	16#4B7A: sMsg := '4B7A function not implemented';
	16#4B7B: sMsg := '4B7B parameter Tangential Following: The radius of the actual circle segment is too small';
	16#4B7C: sMsg := '4B7C parameter FB_NciFeedTablePreparation: pEntry is NULL';
	16#4B7D: sMsg := '4B7D parameter FB_NciFeedTablePreparation: The specified nEntryType does not match the the structure type';
	16#4B7E: sMsg := '4B7E parameter ST_NciMFuncFast and ST_NciMFuncHsk: The requested m-function is not in between 0..159';
	16#4B7F: sMsg := '4B7F parameter ST_NciDynOvr: The requested value for the dynamic override is not in between 0.01 and 1.0';
	16#4B80: sMsg := '4B80 parameter ST_NciVertexSmoothing: invalid parameter. This error occurs with a negative vertex radius or an unknown vertex smoothing type.';
	16#4B81: sMsg := '4B81 parameter FB_NciFeedTablePrepartion: The requested velocity is not in a valid range';
	16#4B82: sMsg := '4B82 parameter ST_Nci*: invalid parameter';

ELSE
	sMsg := UDINT_TO_STRING(iErrID);
	sMsg := concat(sMsg, ' Unknown Error code');
END_CASE
F_AxErrMsg := sMsg;

END_FUNCTION

// ---- POUs/FB/AxisControl/Internal/HomingAdv/FB_HomingLimitSwitch.TcPOU
//==================================================================================================
//							Beckhoff Automation Poland
//									3.01.2022
//	Function block running PLC CAM procedure using hardware limit switch
//	Library: Tc3_MC2_AdvancedHoming, Tc2_MC2, 
//
//  v1.0	|| TC v 3.1.4024.22		|| First edition 
//==================================================================================================
FUNCTION_BLOCK FB_HomingLimitSwitch
VAR_IN_OUT
	Axis 										: Tc2_MC2.AXIS_REF;
END_VAR
VAR_INPUT
	bExecute									: BOOL;
	eDirection									: Tc3_MC2_AdvancedHoming.MC_Home_Direction;
	eLimitSwitchMode							: Tc3_MC2_AdvancedHoming.MC_Switch_Mode;
	eLimitSwitchSignal							: Tc3_MC2_AdvancedHoming.MC_Ref_Signal_Ref;
	lrVelocity									: LREAL;
	lrSetPosition								: LREAL;
	tTimeLimit									: TIME;
	lrDistanceLimit								: LREAL;
	lrTorqueLimit								: LREAL;
	lrDistance									: LREAL;
END_VAR                             		
VAR_OUTPUT                              		
	bDone										: BOOL;
	bBusy										: BOOL;
	bCommandAborted								: BOOL;
	bError										: BOOL;
	nErrorID									: UDINT;
END_VAR
VAR
//=========================== Common ============================
	nStep										: UDINT;
	stParameter									: Tc3_MC2_AdvancedHoming.MC_HomingParameter;
	stOptions									: Tc3_MC2_AdvancedHoming.ST_Home_Options4;
	mcStepLimitSwitch							: Tc3_MC2_AdvancedHoming.MC_StepLimitSwitch;
//=========================== Finish ============================
	mcFinishHoming								: Tc3_MC2_AdvancedHoming.MC_FinishHoming;
//============================ Abort ============================
	mcAbortHoming								: Tc3_MC2_AdvancedHoming.MC_AbortHoming;
//========================== Internal ===========================
    {attribute 'hide'}
	nErrorID_Int								: UDINT;
//===============================================================
END_VAR

//====== Call FBs outside CASE - easier debugging ===============
mcStepLimitSwitch(	Axis						:= Axis, 
					Parameter					:= stParameter,
					LimitSwitchMode				:= eLimitSwitchMode, 
					LimitSwitchSignal			:= eLimitSwitchSignal);
                                        		
mcFinishHoming(	Axis							:= Axis, 
				Parameter						:= stParameter);
				                        	
mcAbortHoming(	Axis							:= Axis, 
				Parameter						:= stParameter);
				
//============== CASE instruction - step machine ================
CASE nStep OF
	
	0: // Wait for command
	
		IF bExecute THEN
			bBusy								:= TRUE;
				
			mcStepLimitSwitch(	Axis			:= Axis, 
								Parameter		:= stParameter,
								Execute			:= TRUE,
								Direction		:= eDirection,  
								Velocity		:= lrVelocity,
								SetPosition		:= lrSetPosition, 
								TimeLimit		:= tTimeLimit, 
								DistanceLimit	:= lrDistanceLimit,
								TorqueLimit		:= lrTorqueLimit,  
								Options			:= stOptions);
								
			// Latch finish parameters
			mcFinishHoming.Distance				:= lrDistance;
			mcFinishHoming.Velocity				:= lrVelocity;
						
			nStep								:= 1000;

		END_IF
	
	1000: // Wait till end
	
		IF mcStepLimitSwitch.Done THEN
			mcStepLimitSwitch.Execute			:= FALSE;
			nStep 								:= 3000;
		END_IF
		
		IF mcStepLimitSwitch.CommandAborted THEN
			mcStepLimitSwitch.Execute			:= FALSE;
			bBusy 								:= FALSE;
			bCommandAborted						:= TRUE;
			nStep 								:= 6000;
		END_IF
		
		IF mcStepLimitSwitch.Error THEN
			mcStepLimitSwitch.Execute			:= FALSE;
			nErrorID_Int						:= mcStepLimitSwitch.ErrorID;
			nStep 								:= 4000;
		END_IF
		
	3000: // MC_FinishHoming
	
		mcFinishHoming.Execute					:= TRUE;				
		nStep									:= nStep + 10;
		
	3010: // Wait till end
	
		IF mcFinishHoming.Done THEN
			mcFinishHoming.Execute				:= FALSE;
			bBusy 								:= FALSE;
			bDone 								:= TRUE;
			nStep 								:= 5000;
		END_IF
		
		IF mcFinishHoming.CommandAborted THEN
			mcFinishHoming.Execute				:= FALSE;
			bBusy 								:= FALSE;
			bCommandAborted						:= TRUE;
			nStep 								:= 6000;
		END_IF
		
		IF mcFinishHoming.Error THEN
			mcFinishHoming.Execute				:= FALSE;
			bBusy 								:= FALSE;
			bError								:= TRUE;
			nErrorID							:= mcFinishHoming.ErrorID;
			nStep 								:= 10000;
		END_IF	
		
	4000: // MC_AbortHoming
	
		mcAbortHoming.Execute					:= TRUE;				
		nStep									:= nStep + 10;
		
	4010: // Wait till end
	
		// No matter what is the end, we go to error State
		IF NOT mcAbortHoming.Busy THEN
			mcAbortHoming.Execute				:= FALSE;
			bBusy 								:= FALSE;
			bError								:= TRUE;
			nErrorID							:= nErrorID_Int;			
			nStep								:= 10000;
		END_IF
		
	5000: // Done
	
		bDone									:= bExecute;
		IF NOT bExecute THEN
			nStep 								:= 0;
		END_IF	
	
	6000: // Command Aborted
	
		bCommandAborted							:= bExecute;
		IF NOT bExecute THEN
			nStep 								:= 0;
		END_IF
		
	10000..20000: // Error
	
		bError									:= bExecute;
		IF NOT bExecute THEN
			nErrorID							:= 0;
			nErrorID_Int						:= 0;
			nStep 								:= 0;
		END_IF
		
END_CASE
//===============================================================

END_FUNCTION_BLOCK

// ---- POUs/FB/AxisControl/Internal/HomingAdv/FB_HomingMemoryAX8000.TcPOU
//==================================================================================================
//							Beckhoff Automation Poland
//									3.01.2022
//	Function block running PLC CAM procedure and writes offset to encoder memory via AX8000
//	During procedure there is need to enable/disable power - external handling needed
//	Velocity to and off cam and moving direction taken from NC Axis settings
//	Library: Tc2_MC2, Tc2_MC2_Drive, Tc2_System
//
//  v1.0	|| TC v 3.1.4024.22		|| First edition 
//==================================================================================================
FUNCTION_BLOCK FB_HomingMemoryAX8000
VAR_IN_OUT                              		
	Axis										: AXIS_REF;
END_VAR  
VAR_INPUT
	bExecute									: BOOL;								// Rising edge executes cmd
	lrPosition									: LREAL;
	eHomingMode									: Tc2_MC2.MC_HomingMode;
	eFeedback									: Tc2_MC2_Drive.E_PositionOffsetFeedback;
	eMemory										: Tc2_MC2_Drive.E_PositionOffsetMemory;
	bCalibrationCam								: BOOL;
	bPowerStatus								: BOOL;								// 
END_VAR                               		
VAR_OUTPUT                              		
	bDone										: BOOL;
	bBusy										: BOOL;
	bCommandAborted								: BOOL;
	bError										: BOOL;
	nErrorID									: UDINT;
	bEnablePower								: BOOL;
END_VAR                                 		
VAR
	// =================================== Local ======================================
	nStep										: DINT;				// Case step
	lrLatchPos									: LREAL;			// Last latched position - cam falling edge
	// ================================ Internal hidden ===============================
    {attribute 'hide'}
	lrPositionMem								: LREAL;
    {attribute 'hide'}
	eHomingModeMem								: Tc2_MC2.MC_HomingMode;
    {attribute 'hide'}
	eFeedbackMem								: Tc2_MC2_Drive.E_PositionOffsetFeedback;
    {attribute 'hide'}
	eMemoryMem									: Tc2_MC2_Drive.E_PositionOffsetMemory;
    {attribute 'hide'}
	lrOffs										: LREAL;
    {attribute 'hide'}
	lrVelocityTw								: LREAL;			// 40xx/6
    {attribute 'hide'}
	lrVelocityOff								: LREAL;			// 40xx/7
    {attribute 'hide'}
	wInvertDirection							: WORD;				// 50xx/101
	// ===================================== FBs ======================================
    {attribute 'hide'}
	fbADSREAD									: ADSREAD;
    {attribute 'hide'}
	mcHome										: MC_Home;
    {attribute 'hide'}
	mcHalt										: MC_Halt;	
    {attribute 'hide'}
	mcReset										: MC_Reset;	
    {attribute 'hide'}
	mcMoveVelocity								: MC_MoveVelocity;
    {attribute 'hide'}
	fbDeletePositionOffset						: FB_CoEAX8000DeletePositionOffset;
    {attribute 'hide'}
	fbSetPositionOffset							: FB_CoEAX8000SetPositionOffset;
	// ================================================================================
END_VAR

fbDeletePositionOffset(Axis:= Axis);
fbSetPositionOffset(Axis:= Axis);
	
mcMoveVelocity(Axis:= Axis);	
mcHalt(Axis:= Axis);
mcHome(Axis := Axis);
mcReset(Axis:= Axis);

CASE nStep OF
	
	0: // Wait for command
	
		IF bExecute THEN
			lrPositionMem						:= lrPosition;
			eHomingModeMem						:= eHomingMode;
			eFeedbackMem						:= eFeedback;
			eMemoryMem							:= eMemory;
			bBusy								:= TRUE;
			nStep 								:= nStep + 10;
		END_IF

	10: // MC_HomingMode.MC_ResetCalibration - All types need it
	
		mcHome.Execute							:= TRUE;
		mcHome.HomingMode						:= MC_HomingMode.MC_ResetCalibration;
		nStep 									:= nStep + 10;

	20: // Wait till end
	
		IF mcHome.Done THEN
			mcHome.Execute						:= FALSE;
			// Next step depends on homing type
			IF eHomingModeMem = MC_HomingMode.MC_ResetCalibration THEN
				bBusy 							:= FALSE;
				bDone							:= TRUE;
				nStep 							:= 5000;
			END_IF
			
			IF eHomingModeMem = MC_HomingMode.MC_DefaultHoming THEN
				nStep							:= 1000;
			END_IF
	
			IF eHomingModeMem = MC_HomingMode.MC_Direct THEN
				nStep							:= 2000;
			END_IF
	
			IF eHomingModeMem = MC_HomingMode.MC_ForceCalibration THEN
				nStep							:= 3000;
			END_IF

		END_IF
		
		IF mcHome.CommandAborted THEN
			mcHome.Execute						:= FALSE;
			bBusy 								:= FALSE;
			bCommandAborted						:= TRUE;
			nStep 								:= 6000;
		END_IF
		
		IF mcHome.Error THEN
			mcHome.Execute						:= FALSE;
			nErrorID							:= mcHome.ErrorID;
			bBusy 								:= FALSE;
			bError								:= TRUE;
			nStep 								:= nStep + 10000;
		END_IF
		
	1000, 2000: // First remove existing position offset

		IF NOT bPowerStatus THEN
			fbDeletePositionOffset.Execute		:= TRUE;
			fbDeletePositionOffset.Feedback		:= eFeedbackMem;
			fbDeletePositionOffset.Memory		:= eMemoryMem;
			nStep 								:= nStep + 10;
		END_IF
		
	1010, 2010: // Wait till command end
	
		IF NOT fbDeletePositionOffset.Busy THEN
			fbDeletePositionOffset.Execute		:= FALSE;
			IF fbDeletePositionOffset.Error THEN
				nErrorID						:= fbDeletePositionOffset.ErrorID;
				bBusy 							:= FALSE;
				bError							:= TRUE;
				nStep 							:= nStep + 10000;
			ELSE
				nStep 							:= nStep + 10;
			END_IF
		END_IF

	1020: // Write 0 offs - to make moves possible
	
		fbSetPositionOffset.Execute				:= TRUE;
		fbSetPositionOffset.Relative			:= TRUE;
		fbSetPositionOffset.Position			:= 0;
		fbSetPositionOffset.Feedback			:= eFeedbackMem;
		fbSetPositionOffset.Memory				:= eMemoryMem;
		nStep 									:= nStep + 10;		
	
	1030:  // Wait till command end
	
		IF NOT fbSetPositionOffset.Busy THEN
			fbSetPositionOffset.Execute		:= FALSE;
			IF fbSetPositionOffset.Error THEN
				nErrorID						:= fbSetPositionOffset.ErrorID;
				bBusy 							:= FALSE;
				bError							:= TRUE;
				nStep 							:= nStep + 10000;
			ELSE
				nStep 							:=  nStep + 10;	
			END_IF
		END_IF

	1040: // Read lrVelocityTw
	
		fbADSREAD(	READ		:= TRUE,
					NETID		:= '', 
					PORT		:= 500,
					IDXGRP		:= 16#4000 + Axis.NcToPlc.AxisId,
					IDXOFFS		:= 16#0006,
					LEN			:= SIZEOF(lrVelocityTw), 
					DESTADDR	:= ADR(lrVelocityTw));
		
		nStep 									:= nStep + 10;

	1060: // Read lrVelocityOff
	
		fbADSREAD(	READ		:= TRUE,
					NETID		:= '', 
					PORT		:= 500,
					IDXGRP		:= 16#4000 + Axis.NcToPlc.AxisId,
					IDXOFFS		:= 16#0007,
					LEN			:= SIZEOF(lrVelocityOff), 
					DESTADDR	:= ADR(lrVelocityOff));
		
		nStep 									:= nStep + 10;
		
	1080: // Read bInvertDirection
	
		fbADSREAD(	READ		:= TRUE,
					NETID		:= '', 
					PORT		:= 500,
					IDXGRP		:= 16#5000 + Axis.NcToPlc.AxisId,
					IDXOFFS		:= 16#0101,
					LEN			:= SIZEOF(wInvertDirection), 
					DESTADDR	:= ADR(wInvertDirection));
		
		nStep 									:= nStep + 10;
	
	1050,1070,1090:  // Wait till command end
	
		fbADSREAD();
		IF NOT fbADSREAD.BUSY THEN
			IF NOT fbADSREAD.ERR THEN
				fbADSREAD(READ:= FALSE);
				nStep 							:= nStep + 10;
			ELSE
				nErrorID						:= fbADSREAD.ERRID;
				bBusy							:= FALSE;
				bError							:= TRUE;
				fbADSREAD(READ:= FALSE);
				nStep 							:= nStep + 10000;	
			END_IF
		END_IF

	1100: // Reset AX8000 offset error
	
		mcReset.Execute							:= TRUE;
		nStep 									:= nStep + 10;

	1110: // Wait till command end	
	
		IF mcReset.Done THEN
			mcReset.Execute						:= FALSE;
			nStep 								:= nStep + 10;
		END_IF
		
		IF mcReset.Error THEN
			mcReset.Execute						:= FALSE;
			nErrorID							:= mcReset.ErrorID;
			bBusy 								:= FALSE;
			bError								:= TRUE;
			nStep 								:= nStep + 10000;
		END_IF	

	1120: // Enable Power request
	
		bEnablePower							:= TRUE;
		nStep 									:= nStep + 10;
		
	1130: // Power status OK?
	
		IF bPowerStatus THEN
			nStep 								:= nStep + 10;	
		END_IF
	
	1140: // Move velocity to calibration cam
	
		IF wInvertDirection.0 THEN
			mcMoveVelocity.Direction			:= MC_Direction.MC_Negative_Direction;
		ELSE
			mcMoveVelocity.Direction			:= MC_Direction.MC_Positive_Direction;
		END_IF
		mcMoveVelocity.Velocity					:= lrVelocityTw;
		mcMoveVelocity.Execute					:= TRUE;
		nStep 									:= nStep + 10;
	
	1150: // Wait till calibration cam rising edge 
	
		IF bCalibrationCam THEN
			mcMoveVelocity.Execute				:= FALSE;
			nStep 								:= nStep + 10;
		END_IF
		
		IF mcMoveVelocity.CommandAborted THEN
			mcMoveVelocity.Execute				:= FALSE;
			bBusy 								:= FALSE;
			bCommandAborted						:= TRUE;
			nStep 								:= 6000;
		END_IF
		
		IF mcMoveVelocity.Error THEN
			mcMoveVelocity.Execute				:= FALSE;
			nErrorID							:= mcMoveVelocity.ErrorID;
			bBusy 								:= FALSE;
			bError								:= TRUE;
			nStep 								:= nStep + 10000;
		END_IF

	1160: // Halt
	
		mcHalt.Execute							:= TRUE;
		nStep 									:= nStep + 10;
		
	1170:  // Wait till command end
	
		IF mcHalt.Done THEN
			mcHalt.Execute						:= FALSE;
			nStep 								:= nStep + 10;
		END_IF
		
		IF mcHalt.CommandAborted THEN
			mcHalt.Execute						:= FALSE;
			bBusy 								:= FALSE;
			bCommandAborted						:= TRUE;
			nStep 								:= 6000;
		END_IF
		
		IF mcHalt.Error THEN
			mcHalt.Execute						:= FALSE;
			nErrorID							:= mcHalt.ErrorID;
			bBusy 								:= FALSE;
			bError								:= TRUE;
			nStep 								:= nStep + 10000;
		END_IF
		
	1180: // Reference cam became free too soon - ErrorID: 16979
	
		IF NOT bCalibrationCam THEN
			nErrorID							:= 16979;
			bBusy 								:= FALSE;
			bError								:= TRUE;
			nStep 								:= nStep + 10000;
		ELSE
			nStep 								:= nStep + 10;
		END_IF
	
	1190: // Move velocity off calibration cam
	
		IF wInvertDirection.0 THEN
			mcMoveVelocity.Direction			:= MC_Direction.MC_Positive_Direction;
		ELSE
			mcMoveVelocity.Direction			:= MC_Direction.MC_Negative_Direction;
		END_IF
		mcMoveVelocity.Velocity					:= lrVelocityOff;
		mcMoveVelocity.Execute					:= TRUE;
		nStep 									:= nStep + 10;
	
	1200: // Wait till calibration cam falling edge 
	
		IF NOT bCalibrationCam THEN
			lrLatchPos 							:= Axis.NcToPlc.ActPos;
			mcMoveVelocity.Execute				:= FALSE;
			nStep 								:= nStep + 10;
		END_IF
		
		IF mcMoveVelocity.CommandAborted THEN
			mcMoveVelocity.Execute				:= FALSE;
			bBusy 								:= FALSE;
			bCommandAborted						:= TRUE;
			nStep 								:= 6000;
		END_IF
		
		IF mcMoveVelocity.Error THEN
			mcMoveVelocity.Execute				:= FALSE;
			nErrorID							:= mcMoveVelocity.ErrorID;
			bBusy 								:= FALSE;
			bError								:= TRUE;
			nStep 								:= nStep + 10000;
		END_IF

	1210: // Halt
	
		mcHalt.Execute							:= TRUE;
		nStep 									:= nStep + 10;
		
	1220:  // Wait till command end
	
		IF mcHalt.Done THEN
			mcHalt.Execute						:= FALSE;
			nStep 								:= nStep + 10;
		END_IF
		
		IF mcHalt.CommandAborted THEN
			mcHalt.Execute						:= FALSE;
			bBusy 								:= FALSE;
			bCommandAborted						:= TRUE;
			nStep 								:= 6000;
		END_IF
		
		IF mcHalt.Error THEN
			mcHalt.Execute						:= FALSE;
			nErrorID							:= mcHalt.ErrorID;
			bBusy 								:= FALSE;
			bError								:= TRUE;
			nStep 								:= nStep + 10000;
		END_IF
		
	1230: // Disable Power request
	
		bEnablePower							:= FALSE;
		nStep 									:= nStep + 10;
		
	1240: // Power status OK?
	
		IF NOT bPowerStatus THEN
			nStep 								:= nStep + 10;	
		END_IF		
	
	1250: // Write pos
	
		lrOffs 									:= lrLatchPos - Axis.NcToPlc.ActPos;
		fbSetPositionOffset.Execute				:= TRUE;
		fbSetPositionOffset.Relative			:= FALSE;
		fbSetPositionOffset.Position			:= lrPositionMem - lrOffs;
		fbSetPositionOffset.Feedback			:= eFeedbackMem;
		fbSetPositionOffset.Memory				:= eMemoryMem;
		nStep 									:= nStep + 10;
		
	1260:  // Wait till command end
	
		IF NOT fbSetPositionOffset.Busy THEN
			fbSetPositionOffset.Execute		:= FALSE;
			IF fbSetPositionOffset.Error THEN
				nErrorID						:= fbSetPositionOffset.ErrorID;
				bBusy 							:= FALSE;
				bError							:= TRUE;
				nStep 							:= nStep + 10000;
			ELSE
				nStep 							:= 3000;		// Set home flag
			END_IF
		END_IF
			
	2020: // Write pos
	
		fbSetPositionOffset.Execute				:= TRUE;
		fbSetPositionOffset.Relative			:= FALSE;
		fbSetPositionOffset.Position			:= lrPositionMem;
		fbSetPositionOffset.Feedback			:= eFeedbackMem;
		fbSetPositionOffset.Memory				:= eMemoryMem;
		nStep 									:= nStep + 10;
		
	2030:  // Wait till command end
	
		IF NOT fbSetPositionOffset.Busy THEN
			fbSetPositionOffset.Execute		:= FALSE;
			IF fbSetPositionOffset.Error THEN
				nErrorID						:= fbSetPositionOffset.ErrorID;
				bBusy 							:= FALSE;
				bError							:= TRUE;
				nStep 							:= nStep + 10000;
			ELSE
				nStep 							:= 3000;		// Set home flag
			END_IF
		END_IF
		
	3000: // MC_HomingMode.MC_ForceCalibration
	
		mcHome.Execute							:= TRUE;
		mcHome.HomingMode						:= MC_HomingMode.MC_ForceCalibration;
		nStep 									:= nStep + 10;

	3010: // Wait till end
	
		IF mcHome.Done THEN
			mcHome.Execute						:= FALSE;
			bBusy 								:= FALSE;
			bDone								:= TRUE;
			nStep 								:= 5000;
		END_IF
		
		IF mcHome.CommandAborted THEN
			bBusy 								:= FALSE;
			bCommandAborted						:= TRUE;
			nStep 								:= 6000;
		END_IF
		
		IF mcHome.Error THEN
			nErrorID							:= mcHome.ErrorID;
			bBusy 								:= FALSE;
			bError								:= TRUE;
			nStep 								:= nStep + 10000;
		END_IF
		
	5000: // Done
	
		bDone									:= bExecute;
		IF NOT bExecute THEN
			nStep 								:= 0;
		END_IF
		
	6000: // Command Aborted
	
		bCommandAborted							:= bExecute;
		IF NOT bExecute THEN
			nStep 								:= 0;
		END_IF
		
	10000..20000: // Error
	
		bError									:= bExecute;
		IF NOT bExecute THEN
			nErrorID							:= 0;
			nStep 								:= 0;
		END_IF
		
END_CASE

END_FUNCTION_BLOCK

// ---- POUs/FB/AxisControl/Internal/HomingAdv/FB_HomingTorqueDetectionSensor.TcPOU
//==================================================================================================
//							Beckhoff Automation Poland
//									3.01.2022
//	Function block running home procedure in torque mode detection
//	Additional sensor can be used
//	Avaliable two modes:
//	1. Lag based - bLagBased = TRUE - define lrLagLimit which decides about end of movement
//	2. Torque based - bLagBased = FALSE - define lrTorqueLimit and lrTorqueTolerance which decides about end of movement
//
//	Library: Tc3_MC2_AdvancedHoming, Tc2_MC2, 
//
//  v1.1	|| TC v 3.1.4024.22		|| Comments added
//  v1.0	|| TC v 3.1.4024.22		|| First edition 
//==================================================================================================
FUNCTION_BLOCK FB_HomingTorqueDetectionSensor
VAR_IN_OUT
	Axis 										: Tc2_MC2.AXIS_REF;
END_VAR  
VAR_INPUT
	bExecute									: BOOL;					// The command is executed with a rising edge.
	bLagBased									: BOOL;					// TRUE: MC_StepBlockLagBased, FALSE: MC_StepBlock
	eDirection									: Tc3_MC2_AdvancedHoming.MC_Home_Direction;	// 
	lrVelocity									: LREAL;				// Maximum travel velocity (>0)
	lrSetPosition								: LREAL;				// Position value to which the axis position is to be set. 
	lrDetectionVelocityLimit					: LREAL;				// Velocity that must be fallen below for the time DetectionVelocityTime in order to detect driving against the fixed stop.
	tDetectionVelocityTime						: TIME;					// Time for detecting the velocity undershoot when driving against the fixed stop.
	tTimeLimit									: TIME;					// Exceeding this time leads to the search procedure being aborted.
	lrDistanceLimit								: LREAL;				// Exceeding this distance in relation to the start position leads to the search procedure being aborted.
	lrTorqueLimit								: LREAL;				// The motor torque is limited to this value, in relation to the weight counterbalance that is possibly parameterized in the drive, in order to avoid mechanical damage.
	lrTorqueTolerance							: LREAL;				// Tolerance related to the TorqueLimit within which driving against the fixed stop is detected.
	lrLagLimit									: LREAL;				// Position lag value which, if exceeded, leads to detection of driving against the fixed stop.
	lrDistance									: LREAL;				// Distance by which the axis moves away from the current position.
	bSensor										: BOOL := TRUE;			// App - additional sensor to be sure if we are in right position
	tTimeout									: TIME := T#10S;		// Time till waiting for sensor ends
END_VAR                             		
VAR_OUTPUT                              		
	bDone										: BOOL;
	bBusy										: BOOL;
	bCommandAborted								: BOOL;
	bError										: BOOL;
	nErrorID									: UDINT;
END_VAR
VAR
//=========================== Common ============================
	nStep										: UDINT;
	stParameter									: Tc3_MC2_AdvancedHoming.MC_HomingParameter;
	stOptions									: Tc3_MC2_AdvancedHoming.ST_Home_Options3;
	stOptions2									: Tc3_MC2_AdvancedHoming.ST_Home_Options2;
//========================= Step Block ==========================
	mcStepBlock									: Tc3_MC2_AdvancedHoming.MC_StepBlockDetection ;
	mcStepBlockLag								: Tc3_MC2_AdvancedHoming.MC_StepBlockLagBasedDetection;
//====================== Move Relative ==========================
	mcMoveRelative								: MC_MoveRelative;
//=========================== Finish ============================
	mcHomeDirect								: MC_HomeDirect;
//============================ Abort ============================
	mcAbortHoming								: Tc3_MC2_AdvancedHoming.MC_AbortHoming;
//========================== Internal ===========================
    {attribute 'hide'}
	nErrorID_Int								: UDINT;
    {attribute 'hide'}
	tonWatchdog									: TON;
//===============================================================
END_VAR

//====== Call FBs outside CASE - easier debugging ===============
mcStepBlockLag(Axis								:= Axis, 
				Parameter						:= stParameter);
				                        		
mcStepBlock(	Axis							:= Axis, 
				Parameter						:= stParameter);	

mcMoveRelative(	Axis							:= Axis);
                                        		
mcAbortHoming(	Axis							:= Axis, 
				Parameter						:= stParameter);
				
mcHomeDirect(	Axis							:= Axis, 
				Parameter						:= stParameter);					
				
//============== CASE instruction - step machine ================
CASE nStep OF
	
	0: // Wait for command
	
		IF bExecute THEN
			bBusy								:= TRUE;
			// Latch finish parameters
			mcMoveRelative.Distance				:= lrDistance;
			mcMoveRelative.Velocity				:= lrVelocity;
			mcHomeDirect.SetPosition			:= lrSetPosition;
			mcHomeDirect.Options				:= stOptions2;
			
			IF bLagBased THEN

				mcStepBlockLag(Axis				:= Axis, 
						Parameter				:= stParameter, 
						Execute					:= TRUE, 
						Direction				:= eDirection, 
						Velocity				:= lrVelocity,
						DetectionVelocityLimit	:= lrDetectionVelocityLimit, 
						DetectionVelocityTime	:= tDetectionVelocityTime, 
						TimeLimit				:= tTimeLimit, 
						DistanceLimit			:= lrDistanceLimit, 
						TorqueLimit				:= lrTorqueLimit, 
						LagLimit				:= lrLagLimit, 
						Options					:= stOptions);
				
				nStep							:= 1000;
				
			ELSE

				mcStepBlock(Axis				:= Axis, 
						Parameter				:= stParameter, 
						Execute					:= TRUE, 
						Direction				:= eDirection, 
						Velocity				:= lrVelocity,
						DetectionVelocityLimit	:= lrDetectionVelocityLimit, 
						DetectionVelocityTime	:= tDetectionVelocityTime, 
						TimeLimit				:= tTimeLimit, 
						DistanceLimit			:= lrDistanceLimit, 
						TorqueLimit				:= lrTorqueLimit, 
						TorqueTolerance			:= lrTorqueTolerance, 
						Options					:= stOptions);
						
				nStep							:= 2000;
				
			END_IF
		END_IF
	
	1000: // Wait till end MC_StepBlockLagBasedDetection
	
		IF mcStepBlockLag.Done THEN
			mcStepBlockLag.Execute				:= FALSE;
			nStep 								:= 3000;
		END_IF
		
		IF mcStepBlockLag.CommandAborted THEN
			mcStepBlockLag.Execute				:= FALSE;
			nStep 								:= 6010;
		END_IF
		
		IF mcStepBlockLag.Error THEN
			mcStepBlockLag.Execute				:= FALSE;
			nErrorID_Int						:= mcStepBlockLag.ErrorID;
			nStep 								:= 6110;
		END_IF
	
	2000: // Wait till end MC_StepBlockDetection
	
		IF mcStepBlock.Done THEN
			mcStepBlock.Execute					:= FALSE;
			nStep 								:= 3000;
		END_IF
		
		IF mcStepBlock.CommandAborted THEN
			mcStepBlock.Execute					:= FALSE;
			nStep 								:= 6020;
		END_IF
		
		IF mcStepBlock.Error THEN
			mcStepBlock.Execute					:= FALSE;
			nErrorID_Int						:= mcStepBlock.ErrorID;
			nStep 								:= 6120;
		END_IF
		
	3000:	// Additional app sample - sensor
	
		tonWatchdog(IN := TRUE, PT := tTimeout);
		IF bSensor THEN
			tonWatchdog(IN := FALSE);
			mcHomeDirect.Execute				:= TRUE;
			nStep								:= nStep + 10;
		ELSIF tonWatchdog.Q THEN
			tonWatchdog(IN := FALSE);
			nStep								:= 6130;
		END_IF
		
	3010: // Wait till end MC_HomeDirect
	
		IF mcHomeDirect.Done THEN
			mcHomeDirect.Execute				:= FALSE;
			nStep 								:= 4000;
		END_IF
		
		IF mcHomeDirect.CommandAborted THEN
			mcHomeDirect.Execute				:= FALSE;
			nStep 								:= 6040;
		END_IF
		
		IF mcHomeDirect.Error THEN
			mcHomeDirect.Execute				:= FALSE;
			nErrorID							:= mcHomeDirect.ErrorID;
			nStep 								:= 6140;
		END_IF		

	4000: // MC_MoveRelative
	
		mcMoveRelative.Execute					:= TRUE;			
		nStep									:= nStep + 10;
	
	4010: // Wait till end MC_MoveRelative
	
		IF mcMoveRelative.Done THEN
			mcMoveRelative.Execute				:= FALSE;
			bBusy 								:= FALSE;
			bDone 								:= TRUE;
			nStep								:= 5000;
		END_IF
		
		IF mcMoveRelative.CommandAborted THEN
			mcMoveRelative.Execute				:= FALSE;
			nStep 								:= 6050;
		END_IF
		
		IF mcMoveRelative.Error THEN
			mcMoveRelative.Execute				:= FALSE;
			nErrorID_Int						:= mcMoveRelative.ErrorID;
			nStep 								:= 6150;
		END_IF		

	
	5000: // Done
	
		bDone									:= bExecute;
		IF NOT bExecute THEN
			nStep 								:= 0;
		END_IF
	
	6000..6199: // MC_AbortHoming
	
		mcAbortHoming.Execute					:= TRUE;				
		nStep									:= nStep + 200;
	
	6200..6399: // Wait till end Command Aborted (..200-..299)/Error (..300/399)
	
		// No matter what is the end, we go to Command Aborted/Error State
		IF NOT mcAbortHoming.Busy THEN
			mcAbortHoming.Execute				:= FALSE;
			bBusy 								:= FALSE;
			// Set CA/E flag
			bCommandAborted						:= nStep < 6300;
			bError								:= NOT bCommandAborted;
			
			IF bError THEN
				nErrorID						:= nErrorID_Int;
				nStep							:= nStep + 10000;
			ELSE
				nStep							:= 7000;
			END_IF
		
		END_IF		
	
	7000: // Command Aborted
	
		bCommandAborted							:= bExecute;
		IF NOT bExecute THEN
			nStep 								:= 0;
		END_IF
		
	10000..20000: // Error
	
		bError									:= bExecute;
		IF NOT bExecute THEN
			nErrorID							:= 0;
			nErrorID_Int						:= 0;
			nStep 								:= 0;
		END_IF
		
END_CASE
//===============================================================

END_FUNCTION_BLOCK

// ---- POUs/FB/AxisControl/Internal/HomingAdv/FB_HomingTorque_1.TcPOU
//==================================================================================================
//							Beckhoff Automation Poland
//									3.01.2022
//	Function block running home procedure in torque mode
//	Avaliable two modes:
//	1. Lag based - bLagBased = TRUE - define lrLagLimit which decides about end of movement
//	2. Torque based - bLagBased = FALSE - define lrTorqueLimit and lrTorqueTolerance which decides about end of movement
//
//	Library: Tc3_MC2_AdvancedHoming, Tc2_MC2, 
//
//  v1.0	|| TC v 3.1.4024.22		|| First edition 
//==================================================================================================
FUNCTION_BLOCK FB_HomingTorque_1
VAR_IN_OUT
	Axis 										: Tc2_MC2.AXIS_REF;
END_VAR  
VAR_INPUT
	bExecute									: BOOL;					// The command is executed with a rising edge.
	bLagBased									: BOOL;					// TRUE: MC_StepBlockLagBased, FALSE: MC_StepBlock
	eDirection									: Tc3_MC2_AdvancedHoming.MC_Home_Direction;	// 
	lrVelocity									: LREAL;				// Maximum travel velocity (>0)
	lrSetPosition								: LREAL;				// Position value to which the axis position is to be set. 
	lrDetectionVelocityLimit					: LREAL;				// Velocity that must be fallen below for the time DetectionVelocityTime in order to detect driving against the fixed stop.
	tDetectionVelocityTime						: TIME;					// Time for detecting the velocity undershoot when driving against the fixed stop.
	tTimeLimit									: TIME;					// Exceeding this time leads to the search procedure being aborted.
	lrDistanceLimit								: LREAL;				// Exceeding this distance in relation to the start position leads to the search procedure being aborted.
	lrTorqueLimit								: LREAL;				// The motor torque is limited to this value, in relation to the weight counterbalance that is possibly parameterized in the drive, in order to avoid mechanical damage.
	lrTorqueTolerance							: LREAL;				// Tolerance related to the TorqueLimit within which driving against the fixed stop is detected.
	lrLagLimit									: LREAL;				// Position lag value which, if exceeded, leads to detection of driving against the fixed stop.
	lrDistance									: LREAL;				// Distance by which the axis moves away from the current position.
END_VAR                             		
VAR_OUTPUT                              		
	bDone										: BOOL;
	bBusy										: BOOL;
	bCommandAborted								: BOOL;
	bError										: BOOL;
	nErrorID									: UDINT;
END_VAR
VAR
//=========================== Common ============================
	nStep										: UDINT;
	stParameter									: Tc3_MC2_AdvancedHoming.MC_HomingParameter;
	stOptions									: Tc3_MC2_AdvancedHoming.ST_Home_Options3;
//========================= Step Block ==========================
	mcStepBlock									: Tc3_MC2_AdvancedHoming.MC_StepBlock;
	mcStepBlockLag								: Tc3_MC2_AdvancedHoming.MC_StepBlockLagBased;
//=========================== Finish ============================
	mcFinishHoming								: Tc3_MC2_AdvancedHoming.MC_FinishHoming;
//============================ Abort ============================
	mcAbortHoming								: Tc3_MC2_AdvancedHoming.MC_AbortHoming;
//========================== Internal ===========================
    {attribute 'hide'}
	nErrorID_Int								: UDINT;
//===============================================================
END_VAR

//====== Call FBs outside CASE - easier debugging ===============
mcStepBlockLag(Axis								:= Axis, 
				Parameter						:= stParameter);
				                        		
mcStepBlock(	Axis							:= Axis, 
				Parameter						:= stParameter);	
                                        		
mcFinishHoming(	Axis							:= Axis, 
				Parameter						:= stParameter);
				                        	
mcAbortHoming(	Axis							:= Axis, 
				Parameter						:= stParameter);
				
//============== CASE instruction - step machine ================
CASE nStep OF
	
	0: // Wait for command
	
		IF bExecute THEN
			bBusy								:= TRUE;
			// Latch finish parameters
			mcFinishHoming.Distance				:= lrDistance;
			mcFinishHoming.Velocity				:= lrVelocity;
				
			IF bLagBased THEN

				mcStepBlockLag(Axis				:= Axis, 
						Parameter				:= stParameter, 
						Execute					:= TRUE, 
						Direction				:= eDirection, 
						Velocity				:= lrVelocity,
						SetPosition				:= lrSetPosition, 
						DetectionVelocityLimit	:= lrDetectionVelocityLimit, 
						DetectionVelocityTime	:= tDetectionVelocityTime, 
						TimeLimit				:= tTimeLimit, 
						DistanceLimit			:= lrDistanceLimit, 
						TorqueLimit				:= lrTorqueLimit, 
						LagLimit				:= lrLagLimit, 
						Options					:= stOptions);
				
				nStep							:= 1000;
				
			ELSE

				mcStepBlock(Axis				:= Axis, 
						Parameter				:= stParameter, 
						Execute					:= TRUE, 
						Direction				:= eDirection, 
						Velocity				:= lrVelocity,
						SetPosition				:= lrSetPosition, 
						DetectionVelocityLimit	:= lrDetectionVelocityLimit, 
						DetectionVelocityTime	:= tDetectionVelocityTime, 
						TimeLimit				:= tTimeLimit, 
						DistanceLimit			:= lrDistanceLimit, 
						TorqueLimit				:= lrTorqueLimit, 
						TorqueTolerance			:= lrTorqueTolerance, 
						Options					:= stOptions);
						
				nStep							:= 2000;
				
			END_IF
		END_IF
	
	1000: // Wait till end
	
		IF mcStepBlockLag.Done THEN
			mcStepBlockLag.Execute				:= FALSE;
			nStep 								:= 3000;
		END_IF
		
		IF mcStepBlockLag.CommandAborted THEN
			mcStepBlockLag.Execute				:= FALSE;
			bBusy 								:= FALSE;
			bCommandAborted						:= TRUE;
			nStep 								:= 6000;
		END_IF
		
		IF mcStepBlockLag.Error THEN
			mcStepBlockLag.Execute				:= FALSE;
			nErrorID_Int						:= mcStepBlockLag.ErrorID;
			nStep 								:= 4000;
		END_IF
	
	2000: // Wait till end
	
		IF mcStepBlock.Done THEN
			mcStepBlock.Execute					:= FALSE;
			nStep 								:= 3000;
		END_IF
		
		IF mcStepBlock.CommandAborted THEN
			mcStepBlock.Execute					:= FALSE;
			bBusy 								:= FALSE;
			bCommandAborted						:= TRUE;
			nStep 								:= 6000;
		END_IF
		
		IF mcStepBlock.Error THEN
			mcStepBlock.Execute					:= FALSE;
			nErrorID_Int						:= mcStepBlock.ErrorID;
			nStep 								:= 4000;
		END_IF
		
	3000: // MC_FinishHoming
	
		mcFinishHoming.Execute					:= TRUE;				
		nStep									:= nStep + 10;
		
	3010: // Wait till end
	
		IF mcFinishHoming.Done THEN
			mcFinishHoming.Execute				:= FALSE;
			bBusy 								:= FALSE;
			bDone 								:= TRUE;
			nStep 								:= 5000;
		END_IF
		
		IF mcFinishHoming.CommandAborted THEN
			mcFinishHoming.Execute				:= FALSE;
			bBusy 								:= FALSE;
			bCommandAborted						:= TRUE;
			nStep 								:= 6000;
		END_IF
		
		IF mcFinishHoming.Error THEN
			mcFinishHoming.Execute				:= FALSE;
			bBusy 								:= FALSE;
			bError								:= TRUE;
			nErrorID							:= mcFinishHoming.ErrorID;
			nStep 								:= 10000;
		END_IF	
		
	4000: // MC_AbortHoming
	
		mcAbortHoming.Execute					:= TRUE;				
		nStep									:= nStep + 10;
		
	4010: // Wait till end
	
		// No matter what is the end, we go to error State
		IF NOT mcAbortHoming.Busy THEN
			mcAbortHoming.Execute				:= FALSE;
			bBusy 								:= FALSE;
			bError								:= TRUE;
			nErrorID							:= nErrorID_Int;			
			nStep								:= 10000;
		END_IF
		
	5000: // Done
		
		bDone									:= bExecute;
		IF NOT bExecute THEN
			nStep 								:= 0;
		END_IF	
	
	6000: // Command Aborted
	
		bCommandAborted							:= bExecute;
		IF NOT bExecute THEN
			nStep 								:= 0;
		END_IF
		
	10000..20000: // Error
	
		bError									:= bExecute;
		IF NOT bExecute THEN
			nErrorID							:= 0;
			nErrorID_Int						:= 0;
			nStep 								:= 0;
		END_IF
		
END_CASE
//===============================================================

END_FUNCTION_BLOCK

// ---- POUs/FB/Blinkers/FUN_Beep.TcPOU
FUNCTION FUN_Beep : BOOL
VAR_INPUT
	note:INT;
	duration:INT;
END_VAR
VAR
END_VAR

// NETWORK 1

END_FUNCTION

// ---- POUs/FB/Charts/FB_SimplePulseGenerator.TcPOU
FUNCTION_BLOCK FB_SimplePulseGenerator
VAR_INPUT
	IbGenerate	AT%I*	:	BOOL;
	tPulseLength		:	TIME;		
END_VAR
VAR_OUTPUT
	QbOut		AT%Q*	:	BOOL;
END_VAR
VAR
	ton					:	TON;
	rtIn				:	R_TRIG;
	iCase				:	INT;
END_VAR

rtIn		(	CLK		:=	IbGenerate						);
ton			(	IN		:=	QbOut,	PT	:=	tPulseLength	);

IF (NOT QbOut AND rtIn.Q) THEN
	QbOut										:=	TRUE;
ELSIF (ton.Q) THEN
	QbOut										:=	FALSE;	
END_IF

END_FUNCTION_BLOCK

// ---- POUs/FB/Conversions/ArrayOfReal_To_String.TcPOU
(****************************************************************************************)
(*							Beckhoff Automation Poland									*)
(*							ArrayOfReal_To_String	 v1.2								*)
(*									30.12.2009											*)
(*								v1.2 - dynamiczny rozmiar tablic						*)
(*		Funkcja konwerująca tablicę zmiennych typu REAL na zmienną typu STRING(255)		*)
(*		Zmienne typu REAL oddzielone są znakiem tabulacji ($t)							*)
(*		Powstały napis nie posiada znaku końca linii ($n)								*)
(*		Uwaga!!																			*)
(*		Należy zwrócić uwagę na ilość znaków przypadającą na każdą zmienną typu REAL	*)
(*______________________________________________________________________________________*)

FUNCTION ArrayOfReal_To_String: STRING(255)
VAR_INPUT
	pData: POINTER TO REAL;
	Length : 	UDINT;
END_VAR
VAR
	pos : UDINT;
	bBusy: BOOL;
	sTemp: STRING(7);
	rTemp: REAL;
END_VAR

pos := 1;
REPEAT
	IF pos > Length THEN
		bBusy := FALSE;
	ELSE
		rTemp := pData^;
		sTemp := LREAL_TO_FMTSTR(rTemp,2,TRUE);
		ArrayOfReal_To_String := CONCAT( ArrayOfReal_To_String,CONCAT(sTemp,'$t'));
		pos := pos + 4;
		(* increment pointer *)
		pData := pData+4;
		bBusy := TRUE;
	END_IF
UNTIL  NOT bBusy
END_REPEAT

END_FUNCTION

// ---- POUs/FB/Conversions/arrBOOL16_TO_WORD.TcPOU
(************************************************************************************)
(*							Beckhoff Automation Poland								*)
(*								arrBOOL16_TO_WORD v1.0								*)
(*									15.02.2010										*)
(*		Funkcja tworząca zmienną typu WORD z tablicy 16 zmiennych typu BOOL			*)
(*__________________________________________________________________________________*)
FUNCTION arrBOOL16_TO_WORD : WORD
VAR_INPUT
	aBool16 : ARRAY [0..15] OF BOOL;
END_VAR

arrBOOL16_TO_WORD.0 := aBool16[0];
arrBOOL16_TO_WORD.1 := aBool16[1];
arrBOOL16_TO_WORD.2 := aBool16[2];
arrBOOL16_TO_WORD.3 := aBool16[3];
arrBOOL16_TO_WORD.4 := aBool16[4];
arrBOOL16_TO_WORD.5 := aBool16[5];
arrBOOL16_TO_WORD.6 := aBool16[6];
arrBOOL16_TO_WORD.7 := aBool16[7];
arrBOOL16_TO_WORD.8 := aBool16[8];
arrBOOL16_TO_WORD.9 := aBool16[9];
arrBOOL16_TO_WORD.10 := aBool16[10];
arrBOOL16_TO_WORD.11 := aBool16[11];
arrBOOL16_TO_WORD.12 := aBool16[12];
arrBOOL16_TO_WORD.13 := aBool16[13];
arrBOOL16_TO_WORD.14 := aBool16[14];
arrBOOL16_TO_WORD.15 := aBool16[15];

END_FUNCTION

// ---- POUs/FB/Conversions/arrBOOL8_TO_BYTE.TcPOU
(****************************************************************************************)
(*							Beckhoff Automation Poland									*)
(*								arrBOOL8_TO_BYTE v1.0									*)
(*									15.02.2010											*)
(*		Funkcja tworząca zmienną typu BYTE z tablicy 8 zmiennych typu BOOL				*)
(*______________________________________________________________________________________*)
FUNCTION arrBOOL8_TO_BYTE : BYTE
VAR_INPUT
	aBool8 : ARRAY [0..7] OF BOOL;
END_VAR

arrBOOL8_TO_BYTE.0 := aBool8[0];
arrBOOL8_TO_BYTE.1 := aBool8[1];
arrBOOL8_TO_BYTE.2 := aBool8[2];
arrBOOL8_TO_BYTE.3 := aBool8[3];
arrBOOL8_TO_BYTE.4 := aBool8[4];
arrBOOL8_TO_BYTE.5 := aBool8[5];
arrBOOL8_TO_BYTE.6 := aBool8[6];
arrBOOL8_TO_BYTE.7 := aBool8[7];

END_FUNCTION

// ---- POUs/FB/Conversions/ArrOfInt_To_String.TcPOU
(****************************************************************************************)
(*							Beckhoff Automation Poland									*)
(*								ArrOfInt_To_String	 v1.2								*)
(*								30.12.2009												*)
(*								v1.2 - dynamiczny rozmiar tablic						*)
(*		Funkcja konwerująca tablicę zmiennych typu INT na zmienną typu STRING(255)		*)
(*		Zmienne typu INT oddzielone są znakiem tabulacji ($t)							*)
(*		Powstały napis nie posiada znaku końca linii ($n)								*)
(*______________________________________________________________________________________*)

FUNCTION ArrOfInt_To_String : STRING(255)
VAR_INPUT
	pData: POINTER TO INT;
	Length : 	UDINT;
END_VAR
VAR
	pos : UDINT;
	bBusy: BOOL;
	iTemp: INT;
END_VAR

pos := 1;
REPEAT
	IF pos > Length THEN
		bBusy := FALSE;
	ELSE
		iTemp := pData^;
		ArrOfInt_To_String := CONCAT(ArrOfInt_To_String,CONCAT(INT_TO_STRING(iTemp),'$t'));
		pos := pos + 2;
		(* increment pointer *)
		pData := pData+2;
		bBusy := TRUE;
	END_IF
UNTIL  NOT bBusy
END_REPEAT

END_FUNCTION

// ---- POUs/FB/Conversions/BitOriented/BCD_TO_INT.TcPOU
(********************************************************************************************)
(*							Beckhoff Automation Poland										*)
(*								FB_BCD_TO_INT	 v1.0										*)
(*									26.06.2008												*)
(*		Funkcja zamieniająca liczbę w formacie BCD na wartość typu integer. 	   			*)
(*		Gdy na wejście funkcji zostanie wprowadzona zła wartość funkcja zwróci wartość  -1	*)
(*__________________________________________________________________________________________*)


FUNCTION BCD_TO_INT : INT	(* Funkcja zwraca wartość typu INT*)
VAR_INPUT
	B:BYTE;					(* Zmienna wejściowa typu Byte*)
END_VAR

IF SHR(B,4)>9 OR B-SHL(SHR(B,4),4)>9 THEN
	BCD_TO_INT:=-1;
ELSE
	BCD_TO_INT:=B-SHR(B,4)*6;
END_IF;

END_FUNCTION

// ---- POUs/FB/Conversions/BitOriented/F_1stByteW.TcPOU
(****************************************************************************************)
(*							Beckhoff Automation Poland									*)
(*									F_1stByteW	v1.0									*)
(*									15.02.2010											*)
(*		Funkcja wyciagajaca mniej znaczacy BYTE ze zmiennej typu WORD					*)
(*							 wyjscie typu WORD											*)
(*______________________________________________________________________________________*)
FUNCTION F_1stByteW : WORD
VAR_INPUT
	wIn:	WORD;
END_VAR

F_1stByteW := wIn AND 16#FF;

END_FUNCTION

// ---- POUs/FB/Conversions/BitOriented/F_1stByteWtoB.TcPOU
(****************************************************************************************)
(*							Beckhoff Automation Poland									*)
(*								F_1stByteWtoB v1.0										*)
(*									15.02.2010											*)
(*		Funkcja wyciagajaca mniej znaczacy BYTE ze zmiennej typu WORD					*)
(*							 wyjscie typu BYTE											*)
(*______________________________________________________________________________________*)
FUNCTION F_1stByteWtoB : BYTE
VAR_INPUT
	wIn		:	WORD;
END_VAR

F_1stByteWtoB := WORD_TO_BYTE(wIn AND 16#FF);

END_FUNCTION

// ---- POUs/FB/Conversions/BitOriented/F_2ndByteW.TcPOU
(****************************************************************************************)
(*							Beckhoff Automation Poland									*)
(*								F_2ndByteW v1.0											*)
(*									15.02.2010											*)
(*		Funkcja wyciagajaca bardziej znaczacy BYTE ze zmiennej typu WORD				*)
(*							 wyjscie typu WORD											*)
(*______________________________________________________________________________________*)
FUNCTION F_2ndByteW : WORD
VAR_INPUT
	wIn		:	WORD;
END_VAR

F_2ndByteW := wIn AND 16#FF00;

END_FUNCTION

// ---- POUs/FB/Conversions/BitOriented/F_2ndByteWtoB.TcPOU
(****************************************************************************************)
(*							Beckhoff Automation Poland									*)
(*								F_2ndByteWtoB v1.0										*)
(*									15.02.2010											*)
(*		Funkcja wyciagajaca bardziej znaczacy BYTE ze zmiennej typu WORD				*)
(*							 	wyjscie typu BYTE										*)
(*______________________________________________________________________________________*)
FUNCTION F_2ndByteWtoB : BYTE
VAR_INPUT
	wIn		:	WORD;
END_VAR

F_2ndByteWtoB := WORD_TO_BYTE(SHR(wIn,8));

END_FUNCTION

// ---- POUs/FB/Conversions/BitOriented/F_MaskWord.TcPOU
(****************************************************************************************)
(*							Beckhoff Automation Poland									*)
(*								F_MaskWord v1.0											*)
(*									15.02.2010											*)
(*		Funkcja wyciagajaca  okreslona ilosc Bitow ze ze zmiennej typu WORD				*)
(*							 wyjscie typu WORD											*)
(*______________________________________________________________________________________*)
FUNCTION F_MaskWord : WORD
VAR_INPUT
	wIn	:	WORD; (*Wejscie*)
	wNo	:	WORD; (*Ilosc bitow, zaczynajac od LSB*)
END_VAR

CASE wNo OF
	0:
	F_MaskWord := wIn AND 2#0;
	1:
	F_MaskWord := wIn AND 2#1;
	2:
	F_MaskWord := wIn AND 2#11;
	3:
	F_MaskWord := wIn AND 2#111;
	4:
	F_MaskWord := wIn AND 2#1111;
	5:
	F_MaskWord := wIn AND 2#11111;
	6:
	F_MaskWord := wIn AND 2#111111;
	7:
	F_MaskWord := wIn AND 2#1111111;
	8:
	F_MaskWord := wIn AND 2#11111111;
	9:
	F_MaskWord := wIn AND 2#111111111;
	10:
	F_MaskWord := wIn AND 2#1111111111;
	11:
	F_MaskWord := wIn AND 2#11111111111;
	12:
	F_MaskWord := wIn AND 2#111111111111;
	13:
	F_MaskWord := wIn AND 2#1111111111111;
	14:
	F_MaskWord := wIn AND 2#11111111111111;
	15:
	F_MaskWord := wIn AND 2#111111111111111;
	16:
	F_MaskWord := wIn;
END_CASE

END_FUNCTION

// ---- POUs/FB/Conversions/BitOriented/L_TBConvArrBitsToDword.TcPOU
(****************************************************************************************)
(*							Beckhoff Automation Poland									*)
(*							L_TBConvArrBitsToDword  v1.0								*)
(*									7.04.2009											*)
(*		This function converts array 32 single bits into a value of type ”double word”	*)
(*______________________________________________________________________________________*)
FUNCTION L_TBConvArrBitsToDword : DWORD
VAR_INPUT
	arrBits: ARRAY [0..31] OF BOOL;
END_VAR

L_TBConvArrBitsToDword.0 := arrBits[0];
L_TBConvArrBitsToDword.1 := arrBits[1];
L_TBConvArrBitsToDword.2 := arrBits[2];
L_TBConvArrBitsToDword.3 := arrBits[3];
L_TBConvArrBitsToDword.4 := arrBits[4];
L_TBConvArrBitsToDword.5 := arrBits[5];
L_TBConvArrBitsToDword.6 := arrBits[6];
L_TBConvArrBitsToDword.7 := arrBits[7];
L_TBConvArrBitsToDword.8 := arrBits[8];
L_TBConvArrBitsToDword.9 := arrBits[9];
L_TBConvArrBitsToDword.10 := arrBits[10];
L_TBConvArrBitsToDword.11 := arrBits[11];
L_TBConvArrBitsToDword.12 := arrBits[12];
L_TBConvArrBitsToDword.13 := arrBits[13];
L_TBConvArrBitsToDword.14 := arrBits[14];
L_TBConvArrBitsToDword.15 := arrBits[15];
L_TBConvArrBitsToDword.16 := arrBits[16];
L_TBConvArrBitsToDword.17 := arrBits[17];
L_TBConvArrBitsToDword.18 := arrBits[18];
L_TBConvArrBitsToDword.19 := arrBits[19];
L_TBConvArrBitsToDword.20 := arrBits[20];
L_TBConvArrBitsToDword.21 := arrBits[21];
L_TBConvArrBitsToDword.22 := arrBits[22];
L_TBConvArrBitsToDword.23 := arrBits[23];
L_TBConvArrBitsToDword.24 := arrBits[24];
L_TBConvArrBitsToDword.25 := arrBits[25];
L_TBConvArrBitsToDword.26 := arrBits[26];
L_TBConvArrBitsToDword.27 := arrBits[27];
L_TBConvArrBitsToDword.28 := arrBits[28];
L_TBConvArrBitsToDword.29 := arrBits[29];
L_TBConvArrBitsToDword.30 := arrBits[30];
L_TBConvArrBitsToDword.31 := arrBits[31];

END_FUNCTION

// ---- POUs/FB/Conversions/BitOriented/L_TBConvBitsToByte.TcPOU
(****************************************************************************************)
(*							Beckhoff Automation Poland									*)
(*							L_TBConvBitsToByte 	 v1.0									*)
(*									29.02.2007											*)
(*			This function converts 8 single bit values into a value of type ”byte”		*)
(*______________________________________________________________________________________*)
FUNCTION L_TBConvBitsToByte : BYTE
VAR_INPUT
	bBit0: BOOL;
	bBit1: BOOL;
	bBit2: BOOL;
	bBit3: BOOL;
	bBit4: BOOL;
	bBit5: BOOL;
	bBit6: BOOL;
	bBit7: BOOL;
END_VAR

L_TBConvBitsToByte.0 := bBit0;
L_TBConvBitsToByte.1 := bBit1;
L_TBConvBitsToByte.2 := bBit2;
L_TBConvBitsToByte.3 := bBit3;
L_TBConvBitsToByte.4 := bBit4;
L_TBConvBitsToByte.5 := bBit5;
L_TBConvBitsToByte.6 := bBit6;
L_TBConvBitsToByte.7 := bBit7;

END_FUNCTION

// ---- POUs/FB/Conversions/BitOriented/L_TBConvBitsToDword.TcPOU
(****************************************************************************************)
(*							Beckhoff Automation Poland									*)
(*							L_TBConvBitsToDword  v1.0									*)
(*									29.02.2007											*)
(*		This function converts 32 single bit values into a value of type ”double word”	*)
(*______________________________________________________________________________________*)
FUNCTION L_TBConvBitsToDword : DWORD
VAR_INPUT
	bBit0: BOOL;
	bBit1: BOOL;
	bBit2: BOOL;
	bBit3: BOOL;
	bBit4: BOOL;
	bBit5: BOOL;
	bBit6: BOOL;
	bBit7: BOOL;
	bBit8: BOOL;
	bBit9: BOOL;
	bBit10: BOOL;
	bBit11: BOOL;
	bBit12: BOOL;
	bBit13: BOOL;
	bBit14: BOOL;
	bBit15: BOOL;
	bBit16: BOOL;
	bBit17: BOOL;
	bBit18: BOOL;
	bBit19: BOOL;
	bBit20: BOOL;
	bBit21: BOOL;
	bBit22: BOOL;
	bBit23: BOOL;
	bBit24: BOOL;
	bBit25: BOOL;
	bBit26: BOOL;
	bBit27: BOOL;
	bBit28: BOOL;
	bBit29: BOOL;
	bBit30: BOOL;
	bBit31: BOOL;
END_VAR

L_TBConvBitsToDword.0 := bBit0;
L_TBConvBitsToDword.1 := bBit1;
L_TBConvBitsToDword.2 := bBit2;
L_TBConvBitsToDword.3 := bBit3;
L_TBConvBitsToDword.4 := bBit4;
L_TBConvBitsToDword.5 := bBit5;
L_TBConvBitsToDword.6 := bBit6;
L_TBConvBitsToDword.7 := bBit7;
L_TBConvBitsToDword.8 := bBit8;
L_TBConvBitsToDword.9 := bBit9;
L_TBConvBitsToDword.10 := bBit10;
L_TBConvBitsToDword.11 := bBit11;
L_TBConvBitsToDword.12 := bBit12;
L_TBConvBitsToDword.13 := bBit13;
L_TBConvBitsToDword.14 := bBit14;
L_TBConvBitsToDword.15 := bBit15;
L_TBConvBitsToDword.16 := bBit16;
L_TBConvBitsToDword.17 := bBit17;
L_TBConvBitsToDword.18 := bBit18;
L_TBConvBitsToDword.19 := bBit19;
L_TBConvBitsToDword.20 := bBit20;
L_TBConvBitsToDword.21 := bBit21;
L_TBConvBitsToDword.22 := bBit22;
L_TBConvBitsToDword.23 := bBit23;
L_TBConvBitsToDword.24 := bBit24;
L_TBConvBitsToDword.25 := bBit25;
L_TBConvBitsToDword.26 := bBit26;
L_TBConvBitsToDword.27 := bBit27;
L_TBConvBitsToDword.28 := bBit28;
L_TBConvBitsToDword.29 := bBit29;
L_TBConvBitsToDword.30 := bBit30;
L_TBConvBitsToDword.31 := bBit31;

END_FUNCTION

// ---- POUs/FB/Conversions/BitOriented/L_TBConvBitsToWord.TcPOU
(****************************************************************************************)
(*							Beckhoff Automation Poland									*)
(*							L_TBConvBitsToWord  v1.0									*)
(*									29.02.2007											*)
(*			This function converts 16 single bit values into a value of type ”word”		*)
(*______________________________________________________________________________________*)
FUNCTION L_TBConvBitsToWord : WORD
VAR_INPUT
	bBit0: BOOL;
	bBit1: BOOL;
	bBit2: BOOL;
	bBit3: BOOL;
	bBit4: BOOL;
	bBit5: BOOL;
	bBit6: BOOL;
	bBit7: BOOL;
	bBit8: BOOL;
	bBit9: BOOL;
	bBit10: BOOL;
	bBit11: BOOL;
	bBit12: BOOL;
	bBit13: BOOL;
	bBit14: BOOL;
	bBit15: BOOL;
END_VAR
VAR
END_VAR

L_TBConvBitsToWord.0 := bBit0;
L_TBConvBitsToWord.1 := bBit1;
L_TBConvBitsToWord.2 := bBit2;
L_TBConvBitsToWord.3 := bBit3;
L_TBConvBitsToWord.4 := bBit4;
L_TBConvBitsToWord.5 := bBit5;
L_TBConvBitsToWord.6 := bBit6;
L_TBConvBitsToWord.7 := bBit7;
L_TBConvBitsToWord.8 := bBit8;
L_TBConvBitsToWord.9 := bBit9;
L_TBConvBitsToWord.10 := bBit10;
L_TBConvBitsToWord.11 := bBit11;
L_TBConvBitsToWord.12 := bBit12;
L_TBConvBitsToWord.13 := bBit13;
L_TBConvBitsToWord.14 := bBit14;
L_TBConvBitsToWord.15 := bBit15;

END_FUNCTION

// ---- POUs/FB/Conversions/BitOriented/L_TBConvByteToBits.TcPOU
(****************************************************************************************)
(*							Beckhoff Automation Poland									*)
(*							L_TBConvByteToBits     v1.0									*)
(*									29.02.2007											*)
(*	This FB returns the 8 corresponding bit values for an input value of type ”byte”	*)
(*______________________________________________________________________________________*)
FUNCTION_BLOCK L_TBConvByteToBits
VAR_INPUT
	byInput: BYTE;
END_VAR
VAR_OUTPUT
	bBit0: BOOL;
	bBit1: BOOL;
	bBit2: BOOL;
	bBit3: BOOL;
	bBit4: BOOL;
	bBit5: BOOL;
	bBit6: BOOL;
	bBit7: BOOL;
END_VAR

bBit0 := byInput.0;
bBit1 := byInput.1;
bBit2 := byInput.2;
bBit3 := byInput.3;
bBit4 := byInput.4;
bBit5 := byInput.5;
bBit6 := byInput.6;
bBit7 := byInput.7;

END_FUNCTION_BLOCK

// ---- POUs/FB/Conversions/BitOriented/L_TBConvDwordToArrBits.TcPOU
(****************************************************************************************)
(*							Beckhoff Automation Poland									*)
(*							L_TBConvDwordToArrBits v1.0									*)
(*									7.04.2009											*)
(* 				This F returns the 32 corresponding ARRAY of bit values 				*)
(*					for an input value of type ”double word”							*)
(*______________________________________________________________________________________*)
FUNCTION L_TBConvDwordToArrBits: ARRAY [0..31] OF BOOL
VAR_INPUT
	dwInput: DWORD;
END_VAR

L_TBConvDwordToArrBits[0]:=dwInput.0;
L_TBConvDwordToArrBits[1]:=dwInput.1;
L_TBConvDwordToArrBits[2]:=dwInput.2;
L_TBConvDwordToArrBits[3]:=dwInput.3;
L_TBConvDwordToArrBits[4]:=dwInput.4;
L_TBConvDwordToArrBits[5]:=dwInput.5;
L_TBConvDwordToArrBits[6]:=dwInput.6;
L_TBConvDwordToArrBits[7]:=dwInput.7;
L_TBConvDwordToArrBits[8]:=dwInput.8;
L_TBConvDwordToArrBits[9]:=dwInput.9;
L_TBConvDwordToArrBits[10]:=dwInput.10;
L_TBConvDwordToArrBits[11]:=dwInput.11;
L_TBConvDwordToArrBits[12]:=dwInput.12;
L_TBConvDwordToArrBits[13]:=dwInput.13;
L_TBConvDwordToArrBits[14]:=dwInput.14;
L_TBConvDwordToArrBits[15]:=dwInput.15;
L_TBConvDwordToArrBits[16]:=dwInput.16;
L_TBConvDwordToArrBits[17]:=dwInput.17;
L_TBConvDwordToArrBits[18]:=dwInput.18;
L_TBConvDwordToArrBits[19]:=dwInput.19;
L_TBConvDwordToArrBits[20]:=dwInput.20;
L_TBConvDwordToArrBits[21]:=dwInput.21;
L_TBConvDwordToArrBits[22]:=dwInput.22;
L_TBConvDwordToArrBits[23]:=dwInput.23;
L_TBConvDwordToArrBits[24]:=dwInput.24;
L_TBConvDwordToArrBits[25]:=dwInput.25;
L_TBConvDwordToArrBits[26]:=dwInput.26;
L_TBConvDwordToArrBits[27]:=dwInput.27;
L_TBConvDwordToArrBits[28]:=dwInput.28;
L_TBConvDwordToArrBits[29]:=dwInput.29;
L_TBConvDwordToArrBits[30]:=dwInput.30;
L_TBConvDwordToArrBits[31]:=dwInput.31;

END_FUNCTION

// ---- POUs/FB/Conversions/BitOriented/L_TBConvDwordToBits.TcPOU
(****************************************************************************************)
(*							Beckhoff Automation Poland									*)
(*							L_TBConvDwordToBits v1.0									*)
(*									29.02.2007											*)
(* This FB returns the 32 corresponding bit values for an input value of type ”double word” *)
(*_______________________________________________________________________________________*)
FUNCTION_BLOCK L_TBConvDwordToBits
VAR_INPUT
	dwInput: DWORD;
END_VAR
VAR_OUTPUT
	bBit0: BOOL;
	bBit1: BOOL;
	bBit2: BOOL;
	bBit3: BOOL;
	bBit4: BOOL;
	bBit5: BOOL;
	bBit6: BOOL;
	bBit7: BOOL;
	bBit8: BOOL;
	bBit9: BOOL;
	bBit10: BOOL;
	bBit11: BOOL;
	bBit12: BOOL;
	bBit13: BOOL;
	bBit14: BOOL;
	bBit15: BOOL;
	bBit16: BOOL;
	bBit17: BOOL;
	bBit18: BOOL;
	bBit19: BOOL;
	bBit20: BOOL;
	bBit21: BOOL;
	bBit22: BOOL;
	bBit23: BOOL;
	bBit24: BOOL;
	bBit25: BOOL;
	bBit26: BOOL;
	bBit27: BOOL;
	bBit28: BOOL;
	bBit29: BOOL;
	bBit30: BOOL;
	bBit31: BOOL;
END_VAR
VAR
END_VAR

bBit0:=dwInput.0;
bBit1:=dwInput.1;
bBit2:=dwInput.2;
bBit3:=dwInput.3;
bBit4:=dwInput.4;
bBit5:=dwInput.5;
bBit6:=dwInput.6;
bBit7:=dwInput.7;
bBit8:=dwInput.8;
bBit9:=dwInput.9;
bBit10:=dwInput.10;
bBit11:=dwInput.11;
bBit12:=dwInput.12;
bBit13:=dwInput.13;
bBit14:=dwInput.14;
bBit15:=dwInput.15;
bBit16:=dwInput.16;
bBit17:=dwInput.17;
bBit18:=dwInput.18;
bBit19:=dwInput.19;
bBit20:=dwInput.20;
bBit21:=dwInput.21;
bBit22:=dwInput.22;
bBit23:=dwInput.23;
bBit24:=dwInput.24;
bBit25:=dwInput.25;
bBit26:=dwInput.26;
bBit27:=dwInput.27;
bBit28:=dwInput.28;
bBit29:=dwInput.29;
bBit30:=dwInput.30;
bBit31:=dwInput.31;

END_FUNCTION_BLOCK

// ---- POUs/FB/Conversions/BitOriented/L_TBConvWordToBits.TcPOU
(****************************************************************************************)
(*							Beckhoff Automation Poland									*)
(*							L_TBConvWordToBits v1.0										*)
(*									29.02.2007											*)
(*	This FB returns the 16 corresponding bit values for an input value of type ” word”	*)
(*______________________________________________________________________________________*)
FUNCTION_BLOCK L_TBConvWordToBits
VAR_INPUT
	wInput:WORD;
END_VAR
VAR_OUTPUT
	bBit0: BOOL;
	bBit1: BOOL;
	bBit2: BOOL;
	bBit3: BOOL;
	bBit4: BOOL;
	bBit5: BOOL;
	bBit6: BOOL;
	bBit7: BOOL;
	bBit8: BOOL;
	bBit9: BOOL;
	bBit10: BOOL;
	bBit11: BOOL;
	bBit12: BOOL;
	bBit13: BOOL;
	bBit14: BOOL;
	bBit15: BOOL;
END_VAR
VAR
END_VAR

bBit0:=wInput.0;
bBit1:=wInput.1;
bBit2:=wInput.2;
bBit3:=wInput.3;
bBit4:=wInput.4;
bBit5:=wInput.5;
bBit6:=wInput.6;
bBit7:=wInput.7;
bBit8:=wInput.8;
bBit9:=wInput.9;
bBit10:=wInput.10;
bBit11:=wInput.11;
bBit12:=wInput.12;
bBit13:=wInput.13;
bBit14:=wInput.14;
bBit15:=wInput.15;

END_FUNCTION_BLOCK

// ---- POUs/FB/Conversions/BitOriented/L_TBGetBitOfByte.TcPOU
(****************************************************************************************)
(*							Beckhoff Automation Poland									*)
(*								L_TBGetBitOfByte v1.0									*)
(*									29.02.2007											*)
(*				This function returns the state of a single bit within a ”byte” value	*)
(*______________________________________________________________________________________*)
FUNCTION L_TBGetBitOfByte : BOOL
VAR_INPUT
	byInput: BYTE;
	byBitNr: BYTE;
END_VAR

CASE byBitNr OF
	0:
	L_TBGetBitOfByte := byInput.0;
	1:
	L_TBGetBitOfByte := byInput.1;
	2:
	L_TBGetBitOfByte := byInput.2;
	3:
	L_TBGetBitOfByte := byInput.3;
	4:
	L_TBGetBitOfByte := byInput.4;
	5:
	L_TBGetBitOfByte := byInput.5;
	6:
	L_TBGetBitOfByte := byInput.6;
	7:
	L_TBGetBitOfByte := byInput.7;
END_CASE

END_FUNCTION

// ---- POUs/FB/Conversions/BitOriented/L_TBGetBitOfDword.TcPOU
(****************************************************************************************)
(*							Beckhoff Automation Poland									*)
(*							L_TBGetBitOfDword v1.0										*)
(*									29.02.2007											*)
(*		This function returns the state of a single bit within a ”double word” value	*)
(*______________________________________________________________________________________*)
FUNCTION L_TBGetBitOfDword : BOOL
VAR_INPUT
	dwInput:DWORD;
	byBitNr:BYTE;
END_VAR
VAR
END_VAR

CASE byBitNr OF
	0:
	L_TBGetBitOfDword:=dwInput.0;
	1:
	L_TBGetBitOfDword:=dwInput.1;
	2:
	L_TBGetBitOfDword:=dwInput.2;
	3:
	L_TBGetBitOfDword:=dwInput.3;
	4:
	L_TBGetBitOfDword:=dwInput.4;
	5:
	L_TBGetBitOfDword:=dwInput.5;
	6:
	L_TBGetBitOfDword:=dwInput.6;
	7:
	L_TBGetBitOfDword:=dwInput.7;
	8:
	L_TBGetBitOfDword:=dwInput.8;
	9:
	L_TBGetBitOfDword:=dwInput.9;
	10:
	L_TBGetBitOfDword:=dwInput.10;
	11:
	L_TBGetBitOfDword:=dwInput.11;
	12:
	L_TBGetBitOfDword:=dwInput.12;
	13:
	L_TBGetBitOfDword:=dwInput.13;
	14:
	L_TBGetBitOfDword:=dwInput.14;
	15:
	L_TBGetBitOfDword:=dwInput.15;
	16:
	L_TBGetBitOfDword:=dwInput.16;
	17:
	L_TBGetBitOfDword:=dwInput.17;
	18:
	L_TBGetBitOfDword:=dwInput.18;
	19:
	L_TBGetBitOfDword:=dwInput.19;
	20:
	L_TBGetBitOfDword:=dwInput.20;
	21:
	L_TBGetBitOfDword:=dwInput.21;
	22:
	L_TBGetBitOfDword:=dwInput.22;
	23:
	L_TBGetBitOfDword:=dwInput.23;
	24:
	L_TBGetBitOfDword:=dwInput.24;
	25:
	L_TBGetBitOfDword:=dwInput.25;
	26:
	L_TBGetBitOfDword:=dwInput.26;
	27:
	L_TBGetBitOfDword:=dwInput.27;
	28:
	L_TBGetBitOfDword:=dwInput.28;
	29:
	L_TBGetBitOfDword:=dwInput.29;
	30:
	L_TBGetBitOfDword:=dwInput.30;
	31:
	L_TBGetBitOfDword:=dwInput.31;
END_CASE

END_FUNCTION

// ---- POUs/FB/Conversions/BitOriented/L_TBGetBitOfWord.TcPOU
(****************************************************************************************)
(*							Beckhoff Automation Poland									*)
(*							L_TBGetBitOfWord v1.0										*)
(*									29.02.2007											*)
(*			This function returns the state of a single bit within a ”word” value		*)
(*______________________________________________________________________________________*)
FUNCTION L_TBGetBitOfWord : BOOL
VAR_INPUT
	wInput:WORD;
	byBitNr:BYTE;
END_VAR
VAR
END_VAR

CASE byBitNr OF
	0:
	L_TBGetBitOfWord:=wInput.0;
	1:
	L_TBGetBitOfWord:=wInput.1;
	2:
	L_TBGetBitOfWord:=wInput.2;
	3:
	L_TBGetBitOfWord:=wInput.3;
	4:
	L_TBGetBitOfWord:=wInput.4;
	5:
	L_TBGetBitOfWord:=wInput.5;
	6:
	L_TBGetBitOfWord:=wInput.6;
	7:
	L_TBGetBitOfWord:=wInput.7;
	8:
	L_TBGetBitOfWord:=wInput.8;
	9:
	L_TBGetBitOfWord:=wInput.9;
	10:
	L_TBGetBitOfWord:=wInput.10;
	11:
	L_TBGetBitOfWord:=wInput.11;
	12:
	L_TBGetBitOfWord:=wInput.12;
	13:
	L_TBGetBitOfWord:=wInput.13;
	14:
	L_TBGetBitOfWord:=wInput.14;
	15:
	L_TBGetBitOfWord:=wInput.15;
END_CASE

END_FUNCTION

// ---- POUs/FB/Conversions/BitOriented/L_TBResetBitOfByte.TcPOU
(****************************************************************************************)
(*							Beckhoff Automation Poland									*)
(*							L_TBResetBitOfByte v1.0										*)
(*									29.02.2007											*)
(*				This function resets a single bit in a value of type ”byte” to “0”		*)
(*______________________________________________________________________________________*)
FUNCTION L_TBResetBitOfByte : BYTE
VAR_INPUT
	byInput: BYTE;
	byBitNr: BYTE;
END_VAR

L_TBResetBitOfByte := byInput;
CASE byBitNr OF
	0:
	L_TBResetBitOfByte.0 := FALSE;
	1:
	L_TBResetBitOfByte.1 := FALSE;
	2:
	L_TBResetBitOfByte.2 := FALSE;
	3:
	L_TBResetBitOfByte.3 := FALSE;
	4:
	L_TBResetBitOfByte.4 := FALSE;
	5:
	L_TBResetBitOfByte.5 := FALSE;
	6:
	L_TBResetBitOfByte.6 := FALSE;
	7:
	L_TBResetBitOfByte.7 := FALSE;
END_CASE

END_FUNCTION

// ---- POUs/FB/Conversions/BitOriented/L_TBResetBitOfDword.TcPOU
(****************************************************************************************)
(*							Beckhoff Automation Poland									*)
(*							L_TBResetBitOfDword v1.0									*)
(*									29.02.2007											*)
(*			This function resets a single bit in a value of type ”double word” to “0”	*)
(*______________________________________________________________________________________*)
FUNCTION L_TBResetBitOfDword : DWORD
VAR_INPUT
	dwInput: DWORD;
	byBitNr: BYTE;
END_VAR
VAR
END_VAR

L_TBResetBitOfDword := dwInput;
CASE byBitNr OF
	0:
	L_TBResetBitOfDword.0 := FALSE;
	1:
	L_TBResetBitOfDword.1 := FALSE;
	2:
	L_TBResetBitOfDword.2 := FALSE;
	3:
	L_TBResetBitOfDword.3 := FALSE;
	4:
	L_TBResetBitOfDword.4 := FALSE;
	5:
	L_TBResetBitOfDword.5 := FALSE;
	6:
	L_TBResetBitOfDword.6 := FALSE;
	7:
	L_TBResetBitOfDword.7 := FALSE;
	8:
	L_TBResetBitOfDword.8 := FALSE;
	9:
	L_TBResetBitOfDword.9 := FALSE;
	10:
	L_TBResetBitOfDword.10 := FALSE;
	11:
	L_TBResetBitOfDword.11 := FALSE;
	12:
	L_TBResetBitOfDword.12 := FALSE;
	13:
	L_TBResetBitOfDword.13 := FALSE;
	14:
	L_TBResetBitOfDword.14 := FALSE;
	15:
	L_TBResetBitOfDword.15 := FALSE;
	16:
	L_TBResetBitOfDword.16 := FALSE;
	17:
	L_TBResetBitOfDword.17 := FALSE;
	18:
	L_TBResetBitOfDword.18 := FALSE;
	19:
	L_TBResetBitOfDword.19 := FALSE;
	20:
	L_TBResetBitOfDword.20 := FALSE;
	21:
	L_TBResetBitOfDword.21 := FALSE;
	22:
	L_TBResetBitOfDword.22 := FALSE;
	23:
	L_TBResetBitOfDword.23 := FALSE;
	24:
	L_TBResetBitOfDword.24 := FALSE;
	25:
	L_TBResetBitOfDword.25 := FALSE;
	26:
	L_TBResetBitOfDword.26 := FALSE;
	27:
	L_TBResetBitOfDword.27 := FALSE;
	28:
	L_TBResetBitOfDword.28 := FALSE;
	29:
	L_TBResetBitOfDword.29 := FALSE;
	30:
	L_TBResetBitOfDword.30 := FALSE;
	31:
	L_TBResetBitOfDword.31 := FALSE;
END_CASE

END_FUNCTION

// ---- POUs/FB/Conversions/BitOriented/L_TBResetBitOfWord.TcPOU
(****************************************************************************************)
(*							Beckhoff Automation Poland									*)
(*							L_TBResetBitOfWord v1.0										*)
(*									29.02.2007											*)
(*				This function resets a single bit in a value of type ”word” to “0”		*)
(*______________________________________________________________________________________*)
FUNCTION L_TBResetBitOfWord : WORD
VAR_INPUT
	wInput: WORD;
	byBitNr: BYTE;
END_VAR
VAR
END_VAR

L_TBResetBitOfWord := wInput;
CASE byBitNr OF
	0:
	L_TBResetBitOfWord.0 := FALSE;
	1:
	L_TBResetBitOfWord.1 := FALSE;
	2:
	L_TBResetBitOfWord.2 := FALSE;
	3:
	L_TBResetBitOfWord.3 := FALSE;
	4:
	L_TBResetBitOfWord.4 := FALSE;
	5:
	L_TBResetBitOfWord.5 := FALSE;
	6:
	L_TBResetBitOfWord.6 := FALSE;
	7:
	L_TBResetBitOfWord.7 := FALSE;
	8:
	L_TBResetBitOfWord.8 := FALSE;
	9:
	L_TBResetBitOfWord.9 := FALSE;
	10:
	L_TBResetBitOfWord.10 := FALSE;
	11:
	L_TBResetBitOfWord.11 := FALSE;
	12:
	L_TBResetBitOfWord.12 := FALSE;
	13:
	L_TBResetBitOfWord.13 := FALSE;
	14:
	L_TBResetBitOfWord.14 := FALSE;
	15:
	L_TBResetBitOfWord.15 := FALSE;
END_CASE

END_FUNCTION

// ---- POUs/FB/Conversions/BitOriented/L_TBSetBitOfByte.TcPOU
(****************************************************************************************)
(*							Beckhoff Automation Poland									*)
(*							L_TBSetBitOfByte v1.0										*)
(*									29.02.2007											*)
(*				This function sets a single bit in a value of type ”byte” to “1”		*)
(*______________________________________________________________________________________*)
FUNCTION L_TBSetBitOfByte : BYTE
VAR_INPUT
	byInput: BYTE;
	byBitNr: BYTE;
END_VAR

L_TBSetBitOfByte := byInput;
CASE byBitNr OF
	0:
	L_TBSetBitOfByte.0 := TRUE;
	1:
	L_TBSetBitOfByte.1 := TRUE;
	2:
	L_TBSetBitOfByte.2 := TRUE;
	3:
	L_TBSetBitOfByte.3 := TRUE;
	4:
	L_TBSetBitOfByte.4 := TRUE;
	5:
	L_TBSetBitOfByte.5 := TRUE;
	6:
	L_TBSetBitOfByte.6 := TRUE;
	7:
	L_TBSetBitOfByte.7 := TRUE;
END_CASE

END_FUNCTION

// ---- POUs/FB/Conversions/BitOriented/L_TBSetBitOfDword.TcPOU
(****************************************************************************************)
(*							Beckhoff Automation Poland									*)
(*							L_TBSetBitOfDword v1.0										*)
(*									29.02.2007											*)
(*			This function sets a single bit in a value of type ”double word” to “1”		*)
(*______________________________________________________________________________________*)
FUNCTION L_TBSetBitOfDword : DWORD
VAR_INPUT
	dwInput: DWORD;
	byBitNr: BYTE;
END_VAR
VAR
END_VAR

L_TBSetBitOfDword := dwInput;
CASE byBitNr OF
	0:
	L_TBSetBitOfDword.0 := TRUE;
	1:
	L_TBSetBitOfDword.1 := TRUE;
	2:
	L_TBSetBitOfDword.2 := TRUE;
	3:
	L_TBSetBitOfDword.3 := TRUE;
	4:
	L_TBSetBitOfDword.4 := TRUE;
	5:
	L_TBSetBitOfDword.5 := TRUE;
	6:
	L_TBSetBitOfDword.6 := TRUE;
	7:
	L_TBSetBitOfDword.7 := TRUE;
	8:
	L_TBSetBitOfDword.8 := TRUE;
	9:
	L_TBSetBitOfDword.9 := TRUE;
	10:
	L_TBSetBitOfDword.10 := TRUE;
	11:
	L_TBSetBitOfDword.11 := TRUE;
	12:
	L_TBSetBitOfDword.12 := TRUE;
	13:
	L_TBSetBitOfDword.13 := TRUE;
	14:
	L_TBSetBitOfDword.14 := TRUE;
	15:
	L_TBSetBitOfDword.15 := TRUE;
	16:
	L_TBSetBitOfDword.16 := TRUE;
	17:
	L_TBSetBitOfDword.17 := TRUE;
	18:
	L_TBSetBitOfDword.18 := TRUE;
	19:
	L_TBSetBitOfDword.19 := TRUE;
	20:
	L_TBSetBitOfDword.20 := TRUE;
	21:
	L_TBSetBitOfDword.21 := TRUE;
	22:
	L_TBSetBitOfDword.22 := TRUE;
	23:
	L_TBSetBitOfDword.23 := TRUE;
	24:
	L_TBSetBitOfDword.24 := TRUE;
	25:
	L_TBSetBitOfDword.25 := TRUE;
	26:
	L_TBSetBitOfDword.26 := TRUE;
	27:
	L_TBSetBitOfDword.27 := TRUE;
	28:
	L_TBSetBitOfDword.28 := TRUE;
	29:
	L_TBSetBitOfDword.29 := TRUE;
	30:
	L_TBSetBitOfDword.30 := TRUE;
	31:
	L_TBSetBitOfDword.31 := TRUE;
END_CASE

END_FUNCTION

// ---- POUs/FB/Conversions/BitOriented/L_TBSetBitOfWord.TcPOU
(****************************************************************************************)
(*							Beckhoff Automation Poland									*)
(*							L_TBSetBitOfWord v1.0										*)
(*									29.02.2007											*)
(*				This function sets a single bit in a value of type ”word” to “1”		*)
(*______________________________________________________________________________________*)
FUNCTION L_TBSetBitOfWord : WORD
VAR_INPUT
	wInput: WORD;
	byBitNr: BYTE;
END_VAR
VAR
END_VAR

L_TBSetBitOfWord := wInput;
CASE byBitNr OF
	0:
	L_TBSetBitOfWord.0 := TRUE;
	1:
	L_TBSetBitOfWord.1 := TRUE;
	2:
	L_TBSetBitOfWord.2 := TRUE;
	3:
	L_TBSetBitOfWord.3 := TRUE;
	4:
	L_TBSetBitOfWord.4 := TRUE;
	5:
	L_TBSetBitOfWord.5 := TRUE;
	6:
	L_TBSetBitOfWord.6 := TRUE;
	7:
	L_TBSetBitOfWord.7 := TRUE;
	8:
	L_TBSetBitOfWord.8 := TRUE;
	9:
	L_TBSetBitOfWord.9 := TRUE;
	10:
	L_TBSetBitOfWord.10 := TRUE;
	11:
	L_TBSetBitOfWord.11 := TRUE;
	12:
	L_TBSetBitOfWord.12 := TRUE;
	13:
	L_TBSetBitOfWord.13 := TRUE;
	14:
	L_TBSetBitOfWord.14 := TRUE;
	15:
	L_TBSetBitOfWord.15 := TRUE;
END_CASE

END_FUNCTION

// ---- POUs/FB/Conversions/BitOriented/L_TBSquareWave.TcPOU
(****************************************************************************************)
(*							Beckhoff Automation Poland									*)
(*								L_TBSquareWave v1.0										*)
(*									29.02.2007											*)
(*	This FB can be used to generate a Boolean square wave signal with a variable high/low time *)
(*______________________________________________________________________________________*)
FUNCTION_BLOCK L_TBSquareWave
VAR_INPUT
	bEnable:BOOL;
	wTimeHigh:WORD;
	wTimeLow:WORD;
END_VAR
VAR_OUTPUT
	bOut:BOOL;
END_VAR
VAR
	ton1: TON;
	ton2: TON;
END_VAR

IF bEnable THEN
	ton1(IN:= NOT ton2.Q, PT:=WORD_TO_TIME(wTimeLow));
	bOut:=NOT ton1.Q;
	ton2(IN:=ton1.Q , PT:=WORD_TO_TIME(wTimeHigh));
ELSE
	bOut:=FALSE;
END_IF

END_FUNCTION_BLOCK

// ---- POUs/FB/Conversions/FB_CONCAT_S2040.TcPOU
(****************************************************************************************)
(*							Beckhoff Automation Poland									*)
(*							FB_CONCAT_S2040	 v1.0										*)
(*									24.5.2011											*)
(*				Blok funkcyjny łączący do 8 zmiennych trypu STRING(max 255 znaków)		*)
(*						w jedną zmienną typu ST_STRING_2040								*)
(*______________________________________________________________________________________*)
FUNCTION_BLOCK FB_CONCAT_S2040
VAR_INPUT
	sString1								:	STRING(255);
END_VAR
VAR
	i										:	INT;				(*iterator*)
	k										:	INT;				(*ostatni zaczety string*)
	wLength									:	WORD;				(*dlugosc ostatniego STRINGa*)
END_VAR
VAR_IN_OUT
	VeryLongString							:	ST_STRING_2040;
END_VAR
VAR_OUTPUT
	wIloscWszystkichZnakow					:	WORD;
END_VAR

k:=0;
wLength:=0;
FOR i := 1 TO 8 DO
	IF LEN(VeryLongString[i]) <> 0 THEN
		wLength := INT_TO_WORD(LEN(VeryLongString[i]));
		k := i;
	END_IF
END_FOR
(* Nie bylo jeszce nic wpisane *)
IF k = 0 THEN
	wIloscWszystkichZnakow := INT_TO_WORD(LEN(sString1));
	MEMCPY(ADR(VeryLongString), ADR(sString1), INT_TO_UINT(LEN(sString1)));
ELSE
	wIloscWszystkichZnakow := INT_TO_WORD((k-1)*256+WORD_TO_INT(wLength));
	IF (WORD_TO_INT(wIloscWszystkichZnakow)+LEN(sString1)) > 2047 THEN
		MEMCPY(ADR(VeryLongString)+wIloscWszystkichZnakow, ADR(sString1), 2047 - wIloscWszystkichZnakow );
	ELSE
		MEMCPY(ADR(VeryLongString)+wIloscWszystkichZnakow, ADR(sString1), INT_TO_UINT(LEN(sString1)));
	END_IF
	wIloscWszystkichZnakow := int_to_word(word_to_int(wIloscWszystkichZnakow) + LEN(sString1));
END_IF

END_FUNCTION_BLOCK

// ---- POUs/FB/Conversions/F_4BYTES_TO_REAL.TcPOU
(************************************************************************************)
(*							Beckhoff Automation Poland								*)
(*							F_4BYTES_TO_REAL v1										*)
(*									21.11.2013										*)
(*					Funkcja zamieniająca 4 zmienne typu BYTE na REAL	 			*)
(*__________________________________________________________________________________*)
FUNCTION F_4BYTES_TO_REAL : REAL
VAR_INPUT
	BByte0		: BYTE;
	BByte1		: BYTE;
	BByte2		: BYTE;
	BByte3		: BYTE;
END_VAR
VAR
	dwDword	: DWORD;
END_VAR

dwDword := BByte3 *16#1000000 + BByte2 *16#10000 + BByte1 *16#100 + BByte0;
MEMCPY(ADR(F_4BYTES_TO_REAL),ADR(dwDword), 4);

END_FUNCTION

// ---- POUs/FB/Conversions/F_8BYTES_TO_LREAL.TcPOU
(************************************************************************************)
(*							Beckhoff Automation Poland								*)
(*							F_8BYTES_TO_LREAL v1.0									*)
(*									3.07.2015										*)
(*					Funkcja zamieniająca 8 zmiennych typu BYTE na LREAL 			*)
(*__________________________________________________________________________________*)
FUNCTION F_8BYTES_TO_LREAL : LREAL
VAR_INPUT
	BByte0		: BYTE;
	BByte1		: BYTE;
	BByte2		: BYTE;
	BByte3		: BYTE;
	BByte4		: BYTE;
	BByte5		: BYTE;
	BByte6		: BYTE;
	BByte7		: BYTE;
END_VAR
VAR
	arrByte	: ARRAY [1..8] OF BYTE;
END_VAR

arrByte[1] := BByte0;
arrByte[2] := BByte1;
arrByte[3] := BByte2;
arrByte[4] := BByte3;
arrByte[5] := BByte4;
arrByte[6] := BByte5;
arrByte[7] := BByte6;
arrByte[8] := BByte7;

MEMCPY(ADR(F_8BYTES_TO_LREAL),ADR(arrByte), 8);

END_FUNCTION

// ---- POUs/FB/Conversions/F_BCDToDec.TcPOU
(************************************************************************************)
(*								Beckhoff Automation Poland							*)
(* 									F_BCDToDec v1.0									*)
(* 										26.06.2014									*)
(*					Funkcja konwertujaca BYTE (kod BCD) na BYTE (DEC)				*)
(*__________________________________________________________________________________*)
FUNCTION F_BCDToDec: BYTE
VAR_INPUT
	BIn:BYTE;
END_VAR

CASE ROL(BIn AND 16#F0,4) OF
0:	F_BCDToDec := 00;
1:	F_BCDToDec := 10;
2:	F_BCDToDec := 20;
3:	F_BCDToDec := 30;
4:	F_BCDToDec := 40;
5:	F_BCDToDec := 50;
6:	F_BCDToDec := 60;
7:	F_BCDToDec := 70;
8:	F_BCDToDec := 80;
9:	F_BCDToDec := 90;
ELSE
	;
END_CASE

CASE BIn AND 16#F OF
0..9:	F_BCDToDec := F_BCDToDec + (BIn AND 16#F);
ELSE
	;
END_CASE

END_FUNCTION

// ---- POUs/FB/Conversions/F_CLEAN_S2040.TcPOU
(****************************************************************************************)
(*							Beckhoff Automation Poland									*)
(*								F_CLEAN_S2040	 v1.0									*)
(*									24.5.2011											*)
(*				Funkcja czyszcząca zawartość zmiennej typu ST_STRING_2040				*)
(*______________________________________________________________________________________*)
FUNCTION F_CLEAN_S2040 : ST_STRING_2040
VAR_INPUT
                VeryLongString: ST_STRING_2040;
END_VAR
VAR
                i: INT;                    (*iterator*)
END_VAR

FOR i := 1 TO 8 DO
                VeryLongString[i] := '$N';
END_FOR

END_FUNCTION

// ---- POUs/FB/Conversions/F_Convert_4BBCD_To_Real.TcPOU
(************************************************************************************************)
(*								Beckhoff Automation Poland										*)
(* 									F_Convert_4BBCD_To_Real v1.0								*)
(* 										26.06.2014												*)
(*	Funkcja konwertujaca 4 zmienne typu BYTE (BCD) na REAL - czesto spotykane w protokole M-Bus	*)
(*______________________________________________________________________________________________*)
FUNCTION F_Convert_4BBCD_To_Real : REAL
VAR_INPUT
	Byte1: BYTE; (* LSB *)
	Byte2: BYTE;
	Byte3: BYTE;
	Byte4: BYTE; (* MSB *)
END_VAR

F_Convert_4BBCD_To_Real := udint_to_real(F_BCDToDec(Byte1)*1+F_BCDToDec(Byte2)*100+F_BCDToDec(Byte3)*10000+F_BCDToDec(Byte4)*1000000);

END_FUNCTION

// ---- POUs/FB/Conversions/F_DWORD_TO_REAL.TcPOU
(********************************************************************************)
(*							Beckhoff Automation Poland							*)
(*							F_DWORD_TO_REAL v1									*)
(*									21.11.2013									*)
(*					Funkcja zamieniająca DWORD na REAL				 			*)
(*______________________________________________________________________________*)
FUNCTION F_DWORD_TO_REAL : REAL
VAR_INPUT
	dwDword	: DWORD;
END_VAR

MEMCPY(ADR(F_DWORD_TO_REAL),ADR(dwDword), 4);

END_FUNCTION

// ---- POUs/FB/Conversions/F_Words_to_Real.TcPOU
(********************************************************************************************)
(*							Beckhoff Automation Poland										*)
(*							F_Words_to_Real													*)
(*									12.05.2011												*)
(*			Funkcja składa dwie wartości typu WORD  i zamienia na watrosc typu REAL			*)
(*__________________________________________________________________________________________*)

FUNCTION F_Words_to_Real : REAL
VAR_INPUT
	wUpperWord : WORD;
	wLowerWord :WORD;
END_VAR
VAR
END_VAR

MEMCPY(ADR(F_Words_to_Real),ADR(wUpperWord),2);
MEMCPY(ADR(F_Words_to_Real)+2,ADR(wLowerWord),2);

END_FUNCTION

// ---- POUs/FB/Conversions/GRAYB_TO_WORD.TcPOU
(****************************************************************************************)
(*							Beckhoff Automation Poland									*)
(*							GRAYB_TO_WORD	 v1.0										*)
(*									29.12.2008											*)
(*		Funkcja konwerująca 16 sygnalow typu BOOL tworzacych kod Graya					*)
(*						 na wartosc decymalna typu WORD									*)
(*______________________________________________________________________________________*)
FUNCTION GRAYB_TO_WORD : WORD
VAR_INPUT
	bIn0: BOOL;
	bIn1: BOOL;
	bIn2: BOOL;
	bIn3: BOOL;
	bIn4: BOOL;
	bIn5: BOOL;
	bIn6: BOOL;
	bIn7: BOOL;
	bIn8: BOOL;
	bIn9: BOOL;
	bIn10: BOOL;
	bIn11: BOOL;
	bIn12: BOOL;
	bIn13: BOOL;
	bIn14: BOOL;
	bIn15: BOOL;
END_VAR

GRAYB_TO_WORD.15 := bIn15 XOR 0;
GRAYB_TO_WORD.14 := bIn14 XOR GRAYB_TO_WORD.15;
GRAYB_TO_WORD.13 := bIn13 XOR GRAYB_TO_WORD.14;
GRAYB_TO_WORD.12 := bIn12 XOR GRAYB_TO_WORD.13;
GRAYB_TO_WORD.11 := bIn11 XOR GRAYB_TO_WORD.12;
GRAYB_TO_WORD.10 := bIn10 XOR GRAYB_TO_WORD.11;
GRAYB_TO_WORD.9 := bIn9 XOR GRAYB_TO_WORD.10;
GRAYB_TO_WORD.8 := bIn8 XOR GRAYB_TO_WORD.9;
GRAYB_TO_WORD.7 := bIn7 XOR GRAYB_TO_WORD.8;
GRAYB_TO_WORD.6 := bIn6 XOR GRAYB_TO_WORD.7;
GRAYB_TO_WORD.5 := bIn5 XOR GRAYB_TO_WORD.6;
GRAYB_TO_WORD.4 := bIn4 XOR GRAYB_TO_WORD.5;
GRAYB_TO_WORD.3 := bIn3 XOR GRAYB_TO_WORD.4;
GRAYB_TO_WORD.2 := bIn2 XOR GRAYB_TO_WORD.3;
GRAYB_TO_WORD.1 := bIn1 XOR GRAYB_TO_WORD.2;
GRAYB_TO_WORD.0 := bIn0 XOR GRAYB_TO_WORD.1;

END_FUNCTION

// ---- POUs/FB/Conversions/GRAYW_TO_WORD.TcPOU
(****************************************************************************************)
(*							Beckhoff Automation Poland									*)
(*							GRAYW_TO_WORD	 v1.0										*)
(*									29.12.2008											*)
(*		Funkcja konwerująca wartosc wejsciowa typu WORD zapisana w kodzie Graya			*)
(*						 na wartosc decymalna typu WORD									*)
(*______________________________________________________________________________________*)
FUNCTION GRAYW_TO_WORD : WORD
VAR_INPUT
	wIn:WORD;
END_VAR
VAR
END_VAR

GRAYW_TO_WORD.15 := wIn.15 XOR 0;
GRAYW_TO_WORD.14 := wIn.14 XOR GRAYW_TO_WORD.15;
GRAYW_TO_WORD.13 := wIn.13 XOR GRAYW_TO_WORD.14;
GRAYW_TO_WORD.12 := wIn.12 XOR GRAYW_TO_WORD.13;
GRAYW_TO_WORD.11 := wIn.11 XOR GRAYW_TO_WORD.12;
GRAYW_TO_WORD.10 := wIn.10 XOR GRAYW_TO_WORD.11;
GRAYW_TO_WORD.9 := wIn.9 XOR GRAYW_TO_WORD.10;
GRAYW_TO_WORD.8 := wIn.8 XOR GRAYW_TO_WORD.9;
GRAYW_TO_WORD.7 := wIn.7 XOR GRAYW_TO_WORD.8;
GRAYW_TO_WORD.6 := wIn.6 XOR GRAYW_TO_WORD.7;
GRAYW_TO_WORD.5 := wIn.5 XOR GRAYW_TO_WORD.6;
GRAYW_TO_WORD.4 := wIn.4 XOR GRAYW_TO_WORD.5;
GRAYW_TO_WORD.3 := wIn.3 XOR GRAYW_TO_WORD.4;
GRAYW_TO_WORD.2 := wIn.2 XOR GRAYW_TO_WORD.3;
GRAYW_TO_WORD.1 := wIn.1 XOR GRAYW_TO_WORD.2;
GRAYW_TO_WORD.0 := wIn.0 XOR GRAYW_TO_WORD.1;

END_FUNCTION

// ---- POUs/FB/DateAndTime/FB_SimpleWorkTime.TcPOU
//==================================================================================================
//							Beckhoff Automation Poland
//									30.03.2017
//	Proste zliczanie czasu pracy, podaje czas aktualnego zalaczenia, ostatniego zalaczenia, sumarycznego zalaczenia
// 	v1.0	|| TC v 3.1.4020.32		|| - pierwsza wersja
//==================================================================================================
FUNCTION_BLOCK FB_SimpleWorkTime
VAR_INPUT
	bIn										: BOOL;
	bReset									: BOOL;					// Zerowanie wartosci
END_VAR
VAR_OUTPUT
	tCurrentTime							: TIME;					// Aktualny czas zalaczenia
	tLastTime								: TIME;					// Ostatni czas zalaczenia
	tSummaryTime							: TIME;					// Sumaryczny czas zalaczenia
END_VAR
VAR
	fbTimeMeasure							: FB_TimeMeasureEx;		// Licznik czasu
	tLastSummaryTime						: TIME;					// Zmienna do wewnetrznych przeliczen
END_VAR

fbTimeMeasure(bOn:= bIn, bReset := bReset, tCurrentTime=> tCurrentTime, tLastTime=> tLastTime);
IF bIn THEN
	tSummaryTime 		:= tLastSummaryTime + tCurrentTime;
ELSE
	tLastSummaryTime 	:= tSummaryTime;
END_IF

IF bReset THEN
	tSummaryTime 		:= T#0S;
	tLastSummaryTime 	:= T#0S;
END_IF

END_FUNCTION_BLOCK

// ---- POUs/FB/DateAndTime/FB_TimeMeasureEx.TcPOU
//==================================================================================================
//							Beckhoff Automation Poland
//									30.03.2017
//		Mierzy czas zalaczenia wejscia. Podaje aktualny czas oraz czas ostatniego zalaczenia
//		W porownaniu do FB_TimeMeasure ma wejscie bReset
// 	v1.0 	|| TC v 3.1.4020.32		|| - pierwsza wersja
//==================================================================================================
FUNCTION_BLOCK FB_TimeMeasureEx
VAR_INPUT
	bOn										: BOOL;					// Zliczany sygnal
	bReset									: BOOL;					// Zerowanie wartosci
END_VAR
VAR_OUTPUT
	tCurrentTime							: TIME;
	tLastTime								: TIME;
END_VAR
VAR
	ton1									: TON;
	bOnOld									: BOOL;
END_VAR

IF bOn = FALSE AND bOnOld = TRUE THEN 
	tLastTime := tCurrentTime; 
END_IF
ton1(IN:= bOn, PT:= T#71582m47s295ms, Q=> , ET=> tCurrentTime);
bOnOld 						:= bOn;
IF bReset THEN
	bOnOld					:= FALSE;
	tLastTime				:= T#0S;
	tCurrentTime			:= T#0S;
	ton1(IN:= FALSE);
END_IF

END_FUNCTION_BLOCK

// ---- POUs/FB/DateAndTime/FB_WorktimeCompact.TcPOU
(****************************************************************************************)
(*							Beckhoff Automation Poland									*)
(*								FB_WorktimeCompact v1.0									*)
(*									31.09.2011											*)
(*							Licznik czasu pracy i liczby załaczeń.						*)
(*			Zmienne IN_OUT powinny być przechowywane po zaniku zasilania				*)
(*______________________________________________________________________________________*)
FUNCTION_BLOCK FB_WorktimeCompact
VAR_INPUT
	bIn			:	BOOL;
END_VAR
VAR_IN_OUT
	dwMinutes	: 	DWORD;
	dwCounts	:	DWORD;
END_VAR
VAR
	Timer		:	TON;
	rtMinute	:	R_TRIG;
	i			:	DWORD;
	iOld		:	DWORD;
	rtOn		:	R_TRIG;
END_VAR

(* Wyciągamy sekundy *)
i := TIME_TO_DWORD(Timer.ET) MOD 60000;

IF bIn THEN
	(* Jak działa to sprawdzamy czy się minuta nie przepętliła *)
	rtMinute(CLK:= iOld>i, Q=> );
ELSE
	(* Jak nie działa to sprawdzamy czy było więcej niż 30 s, jak tak to dodamy minutę *)
	rtMinute(CLK:= i>30000, Q=> );
END_IF
(* Timer odliczający czas *)
Timer(IN:=bIn AND NOT Timer.Q ,PT:= T#24h);
(* Przepisanie poprzednich sekund - do wykrycia przepętlenia *)
iOld := i;
(* Dodanie minuty *)
IF rtMinute.Q THEN
	dwMinutes := dwMinutes+1;
END_IF
(* Licznik załaczeń *)
rtOn(CLK:=bIn);
IF rtOn.Q THEN dwCounts := dwCounts+1; END_IF

END_FUNCTION_BLOCK

// ---- POUs/FB/Diagnostics/POUsDiagnosticComponents/Checks/CheckBounds.TcPOU
// Implicitly generated code : DO NOT EDIT
FUNCTION CheckBounds : DINT
VAR_INPUT
	index, lower, upper: DINT;
END_VAR

// Implicitly generated code : Only an Implementation suggestion
IF  index < lower THEN
	CheckBounds := lower;
	gvlChecks.dCheckBounds := gvlChecks.dCheckBounds + 1;
ELSIF  index > upper THEN
	CheckBounds := upper;
	gvlChecks.dCheckBounds := gvlChecks.dCheckBounds + 1;
ELSE  
	CheckBounds := index;
END_IF

END_FUNCTION

// ---- POUs/FB/Diagnostics/POUsDiagnosticComponents/Checks/CheckDivDInt.TcPOU
// Implicitly generated code : DO NOT EDIT
FUNCTION CheckDivDInt : DINT
VAR_INPUT
	divisor:DINT;
END_VAR

// Implicitly generated code : Only an Implementation suggestion
IF divisor = 0 THEN
	CheckDivDInt:=1;
	gvlChecks.dCheckDivDInt := gvlChecks.dCheckDivDInt + 1;
ELSE
	CheckDivDInt:=divisor;
END_IF;

END_FUNCTION

// ---- POUs/FB/Diagnostics/POUsDiagnosticComponents/Checks/CheckDivLInt.TcPOU
// Implicitly generated code : DO NOT EDIT
FUNCTION CheckDivLInt : LINT
VAR_INPUT
	divisor:LINT;
END_VAR

// Implicitly generated code : Only an Implementation suggestion
IF divisor = 0 THEN
	CheckDivLInt:=1;
	gvlChecks.dCheckDivLInt := gvlChecks.dCheckDivLInt + 1;
ELSE
	CheckDivLInt:=divisor;
END_IF;

END_FUNCTION

// ---- POUs/FB/Diagnostics/POUsDiagnosticComponents/Checks/CheckDivLReal.TcPOU
// Implicitly generated code : DO NOT EDIT
FUNCTION CheckDivLReal : LREAL
VAR_INPUT
	divisor:LREAL;
END_VAR

// Implicitly generated code : Only an Implementation suggestion
IF divisor = 0 THEN
	CheckDivLReal:=1;
	gvlChecks.dCheckDivLReal := gvlChecks.dCheckDivLReal + 1;
ELSE
	CheckDivLReal:=divisor;
END_IF;

END_FUNCTION

// ---- POUs/FB/Diagnostics/POUsDiagnosticComponents/Checks/CheckDivReal.TcPOU
// Implicitly generated code : DO NOT EDIT
FUNCTION CheckDivReal : REAL
VAR_INPUT
	divisor:REAL;
END_VAR

// Implicitly generated code : Only an Implementation suggestion
IF divisor = 0 THEN
	CheckDivReal:=1;
	gvlChecks.dCheckDivReal := gvlChecks.dCheckDivReal + 1;
ELSE
	CheckDivReal:=divisor;
END_IF;

END_FUNCTION

// ---- POUs/FB/Diagnostics/POUsDiagnosticComponents/Checks/CheckPointer.TcPOU
// Implicitly generated code : DO NOT EDIT
FUNCTION CheckPointer : POINTER TO BYTE
VAR_INPUT 
	ptToTest : POINTER TO BYTE; // Destination address of the pointer
	iSize : DINT;		        // Size of the type the pointer points to. (e.g: 20 for POINTER TO ARRAY [0..9] OF INT) 
	iGran : DINT;		        // Granularity of the pointer access. This is the size of the biggest non-structured data type in the type the pointer points to. (e.g: 2 for POINTER TO ARRAY [0..9] OF INT)
	bWrite: BOOL;		        // Indicates read or write Access. TRUE = write access.
END_VAR

// No standard way of implementation. Fill your own code here
CheckPointer := ptToTest;

END_FUNCTION

// ---- POUs/FB/Diagnostics/POUsDiagnosticComponents/Checks/CheckRangeSigned.TcPOU
// Implicitly generated code : DO NOT EDIT
FUNCTION CheckRangeSigned : DINT
VAR_INPUT
	value, lower, upper: DINT;
END_VAR

// Implicitly generated code : Only an Implementation suggestion
IF (value < lower) THEN
	CheckRangeSigned := lower;
	gvlChecks.dCheckRangeSigned := gvlChecks.dCheckRangeSigned + 1;
ELSIF(value > upper) THEN
	CheckRangeSigned := upper;
	gvlChecks.dCheckRangeSigned := gvlChecks.dCheckRangeSigned + 1;
ELSE
	CheckRangeSigned := value;
END_IF

END_FUNCTION

// ---- POUs/FB/Diagnostics/POUsDiagnosticComponents/Checks/CheckRangeUnsigned.TcPOU
// Implicitly generated code : DO NOT EDIT
FUNCTION CheckRangeUnsigned : UDINT
VAR_INPUT
	value, lower, upper: UDINT;
END_VAR

// Implicitly generated code : Only an Implementation suggestion
IF (value < lower) THEN
	CheckRangeUnsigned := lower;
	gvlChecks.dCheckRangeUnsigned := gvlChecks.dCheckRangeUnsigned + 1;
ELSIF(value > upper) THEN
	CheckRangeUnsigned := upper;
	gvlChecks.dCheckRangeUnsigned := gvlChecks.dCheckRangeUnsigned + 1;
ELSE
	CheckRangeUnsigned := value;
END_IF

END_FUNCTION

// ---- POUs/FB/FB_BalluffBMP0005.TcPOU
(* Zaleca się ustawienie tolerancji na poziomie 3%. lrOffsetPercentValue := 3*)

FUNCTION_BLOCK FB_BalluffBMP0005
VAR_INPUT
	diSensorMeasurementValue	AT%I*		: DINT;						//IOLink zmienna z czujnika balluff
	lrOffsetPercentValue					: LREAL;					//To jest tolerancja Otwarcia/Zamknięcia (Podajesz w procentach od 1-100 %)
	
	bRecipeChanged							: BOOL;						//Receptura została zmieniona 
	//Kalibracja
	bCalibration							: BOOL;						//Czujnika wymaga kalibracji, żeby przejść w tryb kalibracji musicie bCalibration wystawić na TRUE
	bAcceptOpenCalibrationValue				: BOOL;						//Procedura kalibracji, Operator potwierdza że chwytak jest otwarty. Przepisuję wartość iolink do zmiennej local
	bAcceptCloseCalibrationValue			: BOOL;						//Procedura kalibracji, Operator potwierdza że chwytak złapał butelkę. Przepisuję wartość iolink do zmiennej local.
	
	sStationName							: STRING(200);
	
END_VAR
VAR_OUTPUT
	bSensorClose							: BOOL;						//Wystawia true, gdy chwytak jest otwarty a wartość czujnika iolink mieści się w zakresie tolerancji 
	bSensorOpen								: BOOL;						//Wystawia true, gdy chwytak jest zamknięty a wartość czujnika mieści się w zakresie tolerancji
	bWarning								: BOOL;						//Ostrzeżenie
	sWarningDescription						: STRING(200);				//Opis ostrzeżenia
	sSensorName								: STRING(200);
	iCalibrationState						: INT;						//Aktualny krok kalibracji
	bCalibrationDone						: BOOL;						// Potwierdzenie popranej kalibracji czujnika
END_VAR
VAR
	tonOpenSensor							: TON;
	tonCloseSensor							: TON;
	
	rtRecipeChanged							: R_TRIG;
	rtCalibration							: R_TRIG;
	
	
	lrCalibrationOpenValue					: LREAL;
	lrCalibrationCloseValue					: LREAL;
	bOpen									: BOOL;
	bClose									: BOOL;
END_VAR

ACT_Warnings();
ACT_Calibration();
ACT_Signals();

ACTION ACT_Calibration:
rtCalibration(CLK:= bCalibration);
rtRecipeChanged(CLK:= bRecipeChanged);


IF rtRecipeChanged.Q THEN
	bCalibrationDone				:= FALSE;
	lrCalibrationOpenValue			:= 0;
	lrCalibrationCloseValue			:= 0;
END_IF

IF rtCalibration.Q AND iCalibrationState <> 0 THEN
	bCalibrationDone				:= FALSE;
	lrCalibrationOpenValue			:= 0;
	lrCalibrationCloseValue			:= 0;
	iCalibrationState				:= 10;
END_IF

CASE iCalibrationState OF
	
	0:
		IF rtCalibration.Q THEN
			bCalibrationDone		:= FALSE;
			lrCalibrationOpenValue	:= 0;
			lrCalibrationCloseValue	:= 0;
			iCalibrationState		:= 10;
		END_IF
		
	10:
		IF bAcceptOpenCalibrationValue THEN
			
			lrCalibrationOpenValue	:= diSensorMeasurementValue;
			iCalibrationState		:= 20;
		END_IF
		
	20:
		IF bAcceptCloseCalibrationValue THEN
			
			bCalibrationDone		:= TRUE;
			
			lrCalibrationCloseValue	:= diSensorMeasurementValue;
			iCalibrationState		:= 0;
		END_IF
		
		
END_CASE
END_ACTION

ACTION ACT_Signals:
tonOpenSensor(IN:= bOpen, PT:= T#50MS);
tonCloseSensor(IN:= bClose, PT:=  T#50MS);

IF lrOffsetPercentValue = 0 THEN	
	lrOffsetPercentValue		:= 1;	
END_IF

IF bCalibrationDone THEN

	IF (diSensorMeasurementValue <= lrCalibrationOpenValue + 10000)(*(lrCalibrationOpenValue* (lrOffsetPercentValue/100)))*) AND
	   (diSensorMeasurementValue >= lrCalibrationOpenValue - 10000)(*(lrCalibrationOpenValue* (lrOffsetPercentValue/100)))*) THEN
	
		bOpen					:= TRUE;	   
	   	bSensorOpen				:= tonOpenSensor.Q;//TRUE;
	   
	ELSE
		
		bOpen					:= FALSE;
		bSensorOpen				:= FALSE;
	END_IF
	
	
	
	
	IF ((diSensorMeasurementValue <= lrCalibrationCloseValue + lrOffsetPercentValue)(*(lrCalibrationCloseValue* (lrOffsetPercentValue/100)))*) AND
	   (diSensorMeasurementValue >= lrCalibrationCloseValue - lrOffsetPercentValue)(*(lrCalibrationCloseValue* (lrOffsetPercentValue/100)))*) )OR
		(diSensorMeasurementValue <= - 4692 + 200 AND diSensorMeasurementValue >=  - 4692 - 200) THEN
		
		bClose					:= TRUE;   
	   	bSensorClose			:= tonCloseSensor.Q;//TRUE;
	   
	ELSE
		bClose					:= FALSE;
		bSensorClose			:= FALSE;	
	END_IF

ELSE
	
	bSensorOpen					:= FALSE;
	bSensorClose				:= FALSE;
END_IF
END_ACTION

ACTION ACT_Warnings:

IF NOT bCalibrationDone AND NOT bWarning THEN
	
	bWarning				:= TRUE;
	sWarningDescription		:= 'Czujnik wymaga kalibracji';
	sSensorName				:= sStationName;
END_IF

//Reset warningów
IF bCalibrationDone THEN
	bWarning				:= FALSE;
	sWarningDescription		:= '';
	sSensorName				:= '';
END_IF
END_ACTION

END_FUNCTION_BLOCK

// ---- POUs/FB/FB_CapFeeder_old.TcPOU
(*
Nazwa:			FB_CapFeederV2
Opis:			Sorter nasadek i podajnik nasadek z podnośnikiem JIESANG
Wersja:			v0.1
Data:			2022-07-07
Autor:			DJA
Urzadzenia:		Silnik sortera, podnośnik JIESANG, Wydmuch, czujniki zapełnienia rękawa
Konfiguracja:	
Info:
-poprawiona wersja sortera względem poprzedniej, przerobione na aktualny standard State i RunningState
*)


FUNCTION_BLOCK FB_CapFeeder_old
VAR_INPUT
	
	bEnable						: BOOL;					//Zezowlenie na pracę stacji sprawdzania
	bEStop						: BOOL;					//Stop Awaryjny nieaktywny
	bRun						: BOOL;					//Włączenie sortera nasadek
	bHoming						: BOOL;					//Zezwolenie na wykonanie bazowania i pozycjonowania stacji sprawdzania
	bHeightSet					: BOOL;					// Bit do bazowania stacji na ustaloną wysokość 
	bIgnoreError				: BOOL;					//Ignorowania błędów cyklu pracy
	bReset						: BOOL;					//Reset błędu, jeśli w stanie "eError"
	lrHeightMotorPositionSV		: LREAL;				//Wysokość zadana na której ma znajdować się stacja
	lrMaxHeight					: LREAL;				//Maksymalna wysokość stacji sprawdzania
	lrMinHeight					: LREAL;				//Minimalna wysokość stacji sprawdzania
	bSorterCapSensor 			: BOOL;					// Wejście z czujnika ultradzwiękowego nasadki sortera
	bFullSleeveSensor			: BOOL;					// Wejście przepełnienia rękawa sortera
	bLevelSensor				: BOOL;					// Czujnik poziomu
	bHomingSensor				: BOOL;					// Wejscie czujnika bazowania napedu 
	iTimeDelayOn				: INT; 					//Czas na właczenie silnika sortera po zaniku sygnału przepełnienia z rękawa
	iTimeDelayOff				: INT; 					// Czas na wylączenie silnika sortera po wykryciu sygnału przepełnienia z rękawa sortera
	iTimeToEmptySleeveError		: INT;					// Czas do włączenia alrmu pustego rękawa
	bEngineOK					: BOOL;					//Wejście czujnika zabezpieczenia silnika 
	InEngineVelocityCV 			: UDINT;		
	InEngineSTW 				: UINT; 				// Statusword transportera wejściowo wyjściowego
	IbEngineWcState				: BOOL; 				// Statusword transportera wejściowo wyjściowego
	bHeightMotorEncoderPulse 	: BOOL;					//Sygnał impulsów enkodera siłownika
	rHeightMotorPositionOffset 	: REAL;					//Wysokość bazowania podnośnika
	bManualMovement				: BOOL; 				//Uruchomienie trybu ruchów ręcznych
	udiStationIndex				: UDINT;				// Indywidualny numer stacji
	sStationName				: STRING;				// Nazwa stacji
	
	tGatesFreq					:	TIME;
	
	bSensorInPipe				:	BOOL;				// Czujnik obecnośći flipflopa w rękawie
END_VAR

VAR_OUTPUT
	eState						: E_Station;			// Aktualny stan stacju
	eRunningState				: E_CapFeederState;		// Stan pracy stacji
	eRunningStateBeforeEstop	: E_CapFeederState;  	// Stan przed Estope
	bError						: BOOL;					// Błąd stacji
	udiErrorID					: UDINT;				// Nr blędu przeciągania formatek
	sErrorDescription			: STRING(200);			// Opis błędu
	sErrorDescription2			: STRING(200);			// Opis błędu
	sErrorStationName			: STRING;				// Nazwa stacj
	udiStationID				: UDINT;				// Nr stacji

	lrHeightMotorPositionCV		: LREAL;				//Aktualna pozycja podnośnika stacji
	bHeightMotorUp				: BOOL;					//Sterowanie silnikiem podnośnika  - RUCH W GÓRĘ
	bHeightMotorDown			: BOOL;					//Sterowanie silnikiem podnośnika  - RUCH W DÓŁ
	bSorterEngine 				: BOOL; 				// Sterowanie silnikiem sortera
	QnEngineVelocitySV 			: UDINT; 				// Nastawa prędkości
	QnEngineCTW 				: UINT;  				// Controlword transportera we/wy	
	bSorterAir 					: BOOL; 				// Sterowanie szybkim zaworem wydmuchu
	bHomingNeeded				: BOOL;					// Wymagane ponowne bazowanie (blad podczas bazowania lub stop awaryjny)
	bHomingDone					: BOOL;					// Stacja zbazowana 
	bCycleDone					: BOOL;					// Sygnał o zakończeniu cyklu
	bCycleNotDone				: BOOL;					// Sygnał o niezakończonym cyklu
	tCycleTime					: TIME;	 				// Czas cyklu 
	sWarningDescription			: STRING;
	bWarning1					: BOOL;
	udiWarningID				: UDINT;
	
	bGate1						:	BOOL;	//Szlaban w podajniku nakrętek #1
	bGate2						:	BOOL;	//Szlaban w podajniku nakrętek #2
	
END_VAR

VAR_IN_OUT
	bManualHeightMotorUp		: BOOL;					//Ruch ręczny podnośnika stacji w górę
	bManualHeightMotorDown		: BOOL;					//Ruch ręczny podnośnika stacji w dół
	bManualSorterEngine			: BOOL;					//Ręczne włączenie silnika sortera
	bManualSorterAir			: BOOL;					//Ręczne włączenie zaworu wydmuchu
	
	bManualGate1				:	BOOL;									// Szlaban #1 w rękawe
	bManualGate2				:	BOOL;									// Szlaban #2 w rękawe		
END_VAR

VAR
	i							:	INT;
	aBufferedSensorValue		:	ARRAY[0..50] OF BOOL;	
	iValvesCycleCase			:	INT;
	rtOutSensor					:	R_TRIG;

	// State
	eLastState					: E_Station;			//Stan ogólny bloku
	eLastStateTemp				: E_Station;			//Stan ogólny bloku
	eLastRunningState			: E_CapFeederState;		//Stan podbloku
	eLastRunningStateTemp		: E_CapFeederState;		//Stan podbloku

	fbHeightMotorEncoder		: FB_JiesangActuatorEncoder;				// Blok enkodera podnośnika chwytaka stabilizującego pod zakręcarką	
	bHeightMotorEncoderCounterReset						:BOOL; 				// Sygnał resetu enkodera
	lrLastHeightMotorPositionCV		: LREAL;				// Pozycja podnośnika w poprzednim cyklu programu
	bHeightMotorEncoderHomed	: BOOL;					// Informacja od enkodera że jest zbazowany		
	bStateError					: BOOL;
	
	tofHeightMotorDown			: TOF;					// Opóźnienie ruchu w dół, żeby nie przeciązać rozruchem układu
	rtEncoderHomed				: R_TRIG;				// Bit zakończenia enkodera
		
	tonHeightNoChange			: TON; 					// Timer wykrycia braku ruchu siłownika zmiany wysokości stacji
	tonHeightNoChangeTime		: TON; 					// Timer wykrycia braku ruchu siłownika zmiany wysokości stacji
	
	tonLimitPosMinReachedDelay	: TON;					// Timer osoiągniecia minimalnej wyskości 
	tonLimitPosMaxReachedDelay	: TON;					// Timer osiągnięcia maksymalnej wyskości
	tonSortingEngineOn			: TON;					// Opóźnienie po załączeniu napędu
	tonSortingEngineOff			: TON;					// Opóźnienie wyłączenia napędu
	tonSleeveFullEngineOn		: TON;					// Czas załączenia napędu po wykrciu braku nasadek
	tonEngineBlocked			: TON;					// Zablokowany silnik	
	rtCapSorterSensor			: R_TRIG;				// Triger
	tonTryUnblockWheel			: TON;					// Czas ruchu falownika w drugą stronę
	tofCapFeederSorterCapSensor	: TOF;					// Opóźnienie sygnału z czujnika obecności nasadki ultradzwiek
	tonCapFeederSorterCapSensor	: TON;					// Opóźnienie sygnału z czujnika obecności nasadki ultradźwięk
	tonAirBeforeStart			: TON;					// Czasówka opóźeniani przedmuchu
	tonAirBeforeStart2			: TON;					// Czasówka opóźeniani przedmuchu
	tonAirAfterStop				: TON;					// Czasówka przedmuchu po zatrzymaniu
	tonStoppingTime				: TON;					// Czasówka zbyt długiego zatrzymawania

	
	tonErrorHeightChange		: TON; 					// Timer błędu zacięcia się podnośnika
	tonEmptySleeveError			: TON;					// Timer pustego rękawa
	tonMaxHeightError			: TON;					// Timer ustawienia zbyt dużej wysokości stacji
	tonMinHeightError			: TON;					// Timer ustawienia zbyt małej wysokości stacji
	tonCycleTimer				: TON;					// Czasówka cyklu
	rtrigCycleTimerRead			: R_TRIG;				// Trigger do statystyk cyklu 
	
	tonSorterEngineError: TON;
	tonHomingSensor: TON;
	TimerOn: TON;
	TimerOff: TON;
	bImpOn: BOOL;
	rtCapFeederSorterCapSensor: R_TRIG;
	bBlowDelay: BOOL;
	tonbBlowDelay: TON;
	
	fbInverter: FB_MitsubishiInverter;
	tonInverterError: TON;
	(*Ostrzeżenia*)
	fbbLevelSensor:	FB_InputFilter;
	(*Inne*)	

	tonGates1	:	TON;	//Czasówka dla szlabanów w rękawe
	tonGates2	:	TON;	//Czasówka dla szlabanów w rękawe
	tonGates3	:	TON;	//Czasówka dla szlabanów w rękawe
	tonGates4	:	TON;	//Czasówka dla szlabanów w rękawe

		
	bGates	    :	BOOL;	//Controla szłabanow w rękawe  
	bTryUnblockWheel : BOOL;
	iTryUnblockWheel : INT;
END_VAR

//Wywołanie bloczków od stacji. Ważna jest ich kolejność!!!
ACT_Limits();
ACT_HeightMotor();
ACT_ErrorHandling();

ACT_Signals();
ACT_Control();
ACT_Inverter();
ACT_Statistic();
ACT_Status();
ACT_Warnings();
aStationID();	

lrLastHeightMotorPositionCV:=lrHeightMotorPositionCV;

ACTION ACT_Control:
	(*****Wyłączenie enable*****)
	IF NOT bEnable THEN
		IF eState <> E_Station.eDisabled AND eState <> E_Station.ePreparingToDisable THEN
				eState 				:= E_Station.ePreparingToDisable; 
		END_IF	
	END_IF

	(*****Estop*****)
	IF NOT bEstop  THEN	
		IF eState <> E_Station.eAborted AND eState <> E_Station.eAborting AND eState <> E_Station.eDisabled THEN
				eState 				:= E_Station.eAborting; 
		END_IF
	END_IF


	CASE eState OF
//--------------------------------------------------------------------------------
// Stan maszyny po wyłączeniu i przygotowanie do uruchomienia
	E_Station.eDisabled: 					// Stan nieaktywnosci (Stacja wyłączona) 
	
		IF bEnable THEN
			eState 				:= E_Station.ePreparingToReady; 
		END_IF 
		
//--------------------------------------------------------------------------------
// Stan maszyny po zatrzymaniu awaryjnym   
	E_Station.eAborted: 					// Stan bezpiecznego zatrzymania (po Abortingu) 

		IF bEStop THEN
			eState 				:= E_Station.ePreparingToReady;
		END_IF
		
